(* IEC 61131-3 sources: smart-home/SmartHome/plc (part 2) *)

(* ---- Resource1.gvl ---- *)
(****************************************************************************
**
** Copyright (C) 2021 Francesco Mandracci
** Contact: https://github.com/fmandracci/smart-home
**
** This file is part of the Smart Home Framework.
**
** Commercial License Usage
** Licensees holding valid commercial licenses may use this file in
** accordance with the terms contained in a written agreement
** between you and the copyright owner.
**
** GNU Lesser General Public License Usage
** Alternatively, this file may be used under the terms of the GNU Lesser
** General Public License version 3 as published by the Free Software
** Foundation and appearing in the file LICENSE included in the
** packaging of this file. Please review the following information to
** ensure the GNU Lesser General Public License version 3 requirements
** will be met: https://www.gnu.org/licenses/lgpl-3.0.html.
**
****************************************************************************)

VAR_GLOBAL
    BA_values: ARRAY [1..32] of BOOL;
    BA_masks: ARRAY [1..32] of DWORD := [
        16#00000001,  16#00000002,  16#00000004,  16#00000008,  16#00000010,  16#00000020,  16#00000040,  16#00000080,
        16#00000100,  16#00000200,  16#00000400,  16#00000800,  16#00001000,  16#00002000,  16#00004000,  16#00008000,
        16#00010000,  16#00020000,  16#00040000,  16#00080000,  16#00100000,  16#00200000,  16#00400000,  16#00800000,
        16#01000000,  16#02000000,  16#04000000,  16#08000000,  16#10000000,  16#20000000,  16#40000000,  16#80000000];

END_VAR

(* ---- BA_CheckSensor.st ---- *)
(****************************************************************************
**
** Copyright (C) 2021 Francesco Mandracci
** Contact: https://github.com/fmandracci/smart-home
**
** This file is part of the Smart Home Framework.
**
** Commercial License Usage
** Licensees holding valid commercial licenses may use this file in
** accordance with the terms contained in a written agreement
** between you and the copyright owner.
**
** GNU Lesser General Public License Usage
** Alternatively, this file may be used under the terms of the GNU Lesser
** General Public License version 3 as published by the Free Software
** Foundation and appearing in the file LICENSE included in the
** packaging of this file. Please review the following information to
** ensure the GNU Lesser General Public License version 3 requirements
** will be met: https://www.gnu.org/licenses/lgpl-3.0.html.
**
****************************************************************************)

FUNCTION BA_CheckSensor
#import "Crosstable.gvl"
#import "Resource1.gvl"
VAR_INPUT
	n : UINT;
    konfig : DWORD;
    mask : DWORD;
    PLC_DigIn : BOOL;
END_VAR
VAR_IN_OUT
	ba_ok : UINT;
    all_ok : BOOL;
END_VAR
VAR
	status : UINT;
END_VAR;

	status := ba_ok;

	if PLC_BA_status = ALARM_STATUS_ARMED or PLC_BA_status = ALARM_STATUS_ENABLED
	   or PLC_BA_status = ALARM_STATUS_RINGING or PLC_BA_status = ALARM_STATUS_MUTED then

		(* NB: this function is called only in (ARMED, ENABLED, RINGING, MUTED *)
		if PLC_BA_enabled_sensors >= n then
			if (konfig and mask) <> 0 then
				(* sensor is configured for checking *)

				if PLC_DigIn then
					(* sensor GOOD *)
					if PLC_BA_status = ALARM_STATUS_ARMED then
						status := ALARM_SENSOR_GOOD;
					elsif PLC_BA_status = ALARM_STATUS_ENABLED then
						status := ALARM_SENSOR_GOOD;
					else (* ALARM_STATUS_RINGING or ALARM_STATUS_MUTED *)
						if ba_ok = ALARM_SENSOR_GOOD then
							status := ALARM_SENSOR_GOOD;
						elsif ba_ok = ALARM_SENSOR_NOT_GOOD then
							status := ALARM_SENSOR_WAS_NG;
						else (* ALARM_SENSOR_WAS_NG *)
							status := ALARM_SENSOR_WAS_NG;
						end_if;
					end_if;

				else
					(* sensor NOT GOOD *)
					all_ok := false; (* <--------------------------= *)
					if PLC_BA_status = ALARM_STATUS_ARMED then
						status := ALARM_SENSOR_STILL_NG;
					elsif PLC_BA_status = ALARM_STATUS_ENABLED then
						status := ALARM_SENSOR_NOT_GOOD;
					else (* ALARM_STATUS_RINGING or ALARM_STATUS_MUTED *)
						status := ALARM_SENSOR_NOT_GOOD;
					end_if;
				end_if;
			else
				(* dark grey: sensor is ignored in this bitmask *)
				status := ALARM_SENSOR_IGNORED;
			end_if;
		else
			(* not visible: sensor is not present *)
			status := ALARM_SENSOR_DISABLED;
		end_if;

	end_if;

	if ba_ok <> status then
		ba_ok := status;
	end_if;

END_FUNCTION

(* ---- BA_CheckSensors.st ---- *)
(****************************************************************************
**
** Copyright (C) 2021 Francesco Mandracci
** Contact: https://github.com/fmandracci/smart-home
**
** This file is part of the Smart Home Framework.
**
** Commercial License Usage
** Licensees holding valid commercial licenses may use this file in
** accordance with the terms contained in a written agreement
** between you and the copyright owner.
**
** GNU Lesser General Public License Usage
** Alternatively, this file may be used under the terms of the GNU Lesser
** General Public License version 3 as published by the Free Software
** Foundation and appearing in the file LICENSE included in the
** packaging of this file. Please review the following information to
** ensure the GNU Lesser General Public License version 3 requirements
** will be met: https://www.gnu.org/licenses/lgpl-3.0.html.
**
****************************************************************************)

FUNCTION BA_CheckSensors : BOOL
#import "Crosstable.gvl"
#import "Resource1.gvl"
VAR_INPUT
    index : UINT;
END_VAR
VAR
	mask : UDINT;
	konfig: DWORD;
	all_ok : BOOL;
END_VAR;

	case index of
	ALARM_INDEX_NOTHING: mask := ALARM_MASK_NOTHING;
	ALARM_INDEX_DAYTIME: mask := PLC_BA_daytime_bitmask;
	ALARM_INDEX_NIGHTTIME: mask := PLC_BA_nighttime_bitmask;
	ALARM_INDEX_EVERYTHING: mask := PLC_BA_everything_bitmask;
	else mask := ALARM_MASK_NOTHING;
	end_case;

	konfig := UDINT_TO_DWORD(mask);
	all_ok := true;

    BA_CheckSensor(1 , konfig, 16#00000001, PLC_BA_DigIn_1 , PLC_BA_OK_1 , all_ok);
    BA_CheckSensor(2 , konfig, 16#00000002, PLC_BA_DigIn_2 , PLC_BA_OK_2 , all_ok);
    BA_CheckSensor(3 , konfig, 16#00000004, PLC_BA_DigIn_3 , PLC_BA_OK_3 , all_ok);
    BA_CheckSensor(4 , konfig, 16#00000008, PLC_BA_DigIn_4 , PLC_BA_OK_4 , all_ok);
    BA_CheckSensor(5 , konfig, 16#00000010, PLC_BA_DigIn_5 , PLC_BA_OK_5 , all_ok);
    BA_CheckSensor(6 , konfig, 16#00000020, PLC_BA_DigIn_6 , PLC_BA_OK_6 , all_ok);
    BA_CheckSensor(7 , konfig, 16#00000040, PLC_BA_DigIn_7 , PLC_BA_OK_7 , all_ok);
    BA_CheckSensor(8 , konfig, 16#00000080, PLC_BA_DigIn_8 , PLC_BA_OK_8 , all_ok);
    BA_CheckSensor(9 , konfig, 16#00000100, PLC_BA_DigIn_9 , PLC_BA_OK_9 , all_ok);
    BA_CheckSensor(10, konfig, 16#00000200, PLC_BA_DigIn_10, PLC_BA_OK_10, all_ok);
    BA_CheckSensor(11, konfig, 16#00000400, PLC_BA_DigIn_11, PLC_BA_OK_11, all_ok);
    BA_CheckSensor(12, konfig, 16#00000800, PLC_BA_DigIn_12, PLC_BA_OK_12, all_ok);
    BA_CheckSensor(13, konfig, 16#00001000, PLC_BA_DigIn_13, PLC_BA_OK_13, all_ok);
    BA_CheckSensor(14, konfig, 16#00002000, PLC_BA_DigIn_14, PLC_BA_OK_14, all_ok);
    BA_CheckSensor(15, konfig, 16#00004000, PLC_BA_DigIn_15, PLC_BA_OK_15, all_ok);
    BA_CheckSensor(16, konfig, 16#00008000, PLC_BA_DigIn_16, PLC_BA_OK_16, all_ok);

    BA_CheckSensor(17, konfig, 16#00010000, PLC_BA_DigIn_17, PLC_BA_OK_17, all_ok);
    BA_CheckSensor(18, konfig, 16#00020000, PLC_BA_DigIn_18, PLC_BA_OK_18, all_ok);
    BA_CheckSensor(19, konfig, 16#00040000, PLC_BA_DigIn_19, PLC_BA_OK_19, all_ok);
    BA_CheckSensor(20, konfig, 16#00080000, PLC_BA_DigIn_20, PLC_BA_OK_20, all_ok);
    BA_CheckSensor(21, konfig, 16#00100000, PLC_BA_DigIn_21, PLC_BA_OK_21, all_ok);
    BA_CheckSensor(22, konfig, 16#00200000, PLC_BA_DigIn_22, PLC_BA_OK_22, all_ok);
    BA_CheckSensor(23, konfig, 16#00400000, PLC_BA_DigIn_23, PLC_BA_OK_23, all_ok);
    BA_CheckSensor(24, konfig, 16#00800000, PLC_BA_DigIn_24, PLC_BA_OK_24, all_ok);
    BA_CheckSensor(25, konfig, 16#01000000, PLC_BA_DigIn_25, PLC_BA_OK_25, all_ok);
    BA_CheckSensor(26, konfig, 16#02000000, PLC_BA_DigIn_26, PLC_BA_OK_26, all_ok);
    BA_CheckSensor(27, konfig, 16#04000000, PLC_BA_DigIn_27, PLC_BA_OK_27, all_ok);
    BA_CheckSensor(28, konfig, 16#08000000, PLC_BA_DigIn_28, PLC_BA_OK_28, all_ok);
    BA_CheckSensor(29, konfig, 16#10000000, PLC_BA_DigIn_29, PLC_BA_OK_29, all_ok);
    BA_CheckSensor(30, konfig, 16#20000000, PLC_BA_DigIn_30, PLC_BA_OK_30, all_ok);
    BA_CheckSensor(31, konfig, 16#40000000, PLC_BA_DigIn_31, PLC_BA_OK_31, all_ok);
    BA_CheckSensor(32, konfig, 16#80000000, PLC_BA_DigIn_32, PLC_BA_OK_32, all_ok);

	BA_CheckSensors := all_ok;

END_FUNCTION

(* ---- BA_ClearOK.st ---- *)
(****************************************************************************
**
** Copyright (C) 2021 Francesco Mandracci
** Contact: https://github.com/fmandracci/smart-home
**
** This file is part of the Smart Home Framework.
**
** Commercial License Usage
** Licensees holding valid commercial licenses may use this file in
** accordance with the terms contained in a written agreement
** between you and the copyright owner.
**
** GNU Lesser General Public License Usage
** Alternatively, this file may be used under the terms of the GNU Lesser
** General Public License version 3 as published by the Free Software
** Foundation and appearing in the file LICENSE included in the
** packaging of this file. Please review the following information to
** ensure the GNU Lesser General Public License version 3 requirements
** will be met: https://www.gnu.org/licenses/lgpl-3.0.html.
**
****************************************************************************)

FUNCTION BA_ClearOK : UINT
#import "Crosstable.gvl"
#import "Resource1.gvl"
VAR_INPUT
    n : UINT;
END_VAR

	if PLC_BA_enabled_sensors >= n then
		BA_ClearOK := ALARM_SENSOR_IGNORED;
	else
		BA_ClearOK := ALARM_SENSOR_DISABLED;
	end_if;

END_FUNCTION

(* ---- BA_ClearOKs.st ---- *)
(****************************************************************************
**
** Copyright (C) 2021 Francesco Mandracci
** Contact: https://github.com/fmandracci/smart-home
**
** This file is part of the Smart Home Framework.
**
** Commercial License Usage
** Licensees holding valid commercial licenses may use this file in
** accordance with the terms contained in a written agreement
** between you and the copyright owner.
**
** GNU Lesser General Public License Usage
** Alternatively, this file may be used under the terms of the GNU Lesser
** General Public License version 3 as published by the Free Software
** Foundation and appearing in the file LICENSE included in the
** packaging of this file. Please review the following information to
** ensure the GNU Lesser General Public License version 3 requirements
** will be met: https://www.gnu.org/licenses/lgpl-3.0.html.
**
****************************************************************************)

FUNCTION BA_ClearOKs
#import "Crosstable.gvl"
#import "Resource1.gvl"

    PLC_BA_OK_1  := BA_ClearOK(1 );
    PLC_BA_OK_2  := BA_ClearOK(2 );
    PLC_BA_OK_3  := BA_ClearOK(3 );
    PLC_BA_OK_4  := BA_ClearOK(4 );
    PLC_BA_OK_5  := BA_ClearOK(5 );
    PLC_BA_OK_6  := BA_ClearOK(6 );
    PLC_BA_OK_7  := BA_ClearOK(7 );
    PLC_BA_OK_8  := BA_ClearOK(8 );
    PLC_BA_OK_9  := BA_ClearOK(9 );
    PLC_BA_OK_10 := BA_ClearOK(10);
    PLC_BA_OK_11 := BA_ClearOK(11);
    PLC_BA_OK_12 := BA_ClearOK(12);
    PLC_BA_OK_13 := BA_ClearOK(13);
    PLC_BA_OK_14 := BA_ClearOK(14);
    PLC_BA_OK_15 := BA_ClearOK(15);
    PLC_BA_OK_16 := BA_ClearOK(16);

    PLC_BA_OK_17 := BA_ClearOK(17);
    PLC_BA_OK_18 := BA_ClearOK(18);
    PLC_BA_OK_19 := BA_ClearOK(19);
    PLC_BA_OK_20 := BA_ClearOK(20);
    PLC_BA_OK_21 := BA_ClearOK(21);
    PLC_BA_OK_22 := BA_ClearOK(22);
    PLC_BA_OK_23 := BA_ClearOK(23);
    PLC_BA_OK_24 := BA_ClearOK(24);
    PLC_BA_OK_25 := BA_ClearOK(25);
    PLC_BA_OK_26 := BA_ClearOK(26);
    PLC_BA_OK_27 := BA_ClearOK(27);
    PLC_BA_OK_28 := BA_ClearOK(28);
    PLC_BA_OK_29 := BA_ClearOK(29);
    PLC_BA_OK_30 := BA_ClearOK(30);
    PLC_BA_OK_31 := BA_ClearOK(31);
    PLC_BA_OK_32 := BA_ClearOK(32);

END_FUNCTION

(* ---- BA_ReadSensor.st ---- *)
(****************************************************************************
**
** Copyright (C) 2021 Francesco Mandracci
** Contact: https://github.com/fmandracci/smart-home
**
** This file is part of the Smart Home Framework.
**
** Commercial License Usage
** Licensees holding valid commercial licenses may use this file in
** accordance with the terms contained in a written agreement
** between you and the copyright owner.
**
** GNU Lesser General Public License Usage
** Alternatively, this file may be used under the terms of the GNU Lesser
** General Public License version 3 as published by the Free Software
** Foundation and appearing in the file LICENSE included in the
** packaging of this file. Please review the following information to
** ensure the GNU Lesser General Public License version 3 requirements
** will be met: https://www.gnu.org/licenses/lgpl-3.0.html.
**
****************************************************************************)

FUNCTION BA_ReadSensor : BOOL
#import "Crosstable.gvl"
#import "Resource1.gvl"
VAR_INPUT
    n : UINT;
END_VAR

	if PLC_BA_enabled_sensors >= n then

		if PLC_control_type = ControlType_2 then
			(* MPNE_A, MPNE_B on RTU0 *)
			if n <= 16 then
				if NODE_11_STATUS = NODE_NODE_OK then
					case n of
		             1: SetMpneDigDir_IN(MPNE_A_DigDir_1); BA_ReadSensor := MPNE_A_DigIn_1 ;
		             2: SetMpneDigDir_IN(MPNE_A_DigDir_2); BA_ReadSensor := MPNE_A_DigIn_2 ;
		             3: SetMpneDigDir_IN(MPNE_A_DigDir_3); BA_ReadSensor := MPNE_A_DigIn_3 ;
		             4: SetMpneDigDir_IN(MPNE_A_DigDir_4); BA_ReadSensor := MPNE_A_DigIn_4 ;
		             5: SetMpneDigDir_IN(MPNE_A_DigDir_5); BA_ReadSensor := MPNE_A_DigIn_5 ;
		             6: SetMpneDigDir_IN(MPNE_A_DigDir_6); BA_ReadSensor := MPNE_A_DigIn_6 ;
		             7: SetMpneDigDir_IN(MPNE_A_DigDir_7); BA_ReadSensor := MPNE_A_DigIn_7 ;
		             8: SetMpneDigDir_IN(MPNE_A_DigDir_8); BA_ReadSensor := MPNE_A_DigIn_8 ;
		             9:                                    BA_ReadSensor := MPNE_A_DigIn_9 ;
		            10:                                    BA_ReadSensor := MPNE_A_DigIn_10;
		            11:                                    BA_ReadSensor := MPNE_A_DigIn_11;
		            12:                                    BA_ReadSensor := MPNE_A_DigIn_12;
		            13:                                    BA_ReadSensor := MPNE_A_DigIn_13;
		            14:                                    BA_ReadSensor := MPNE_A_DigIn_14;
		            15:                                    BA_ReadSensor := MPNE_A_DigIn_15;
		            16:                                    BA_ReadSensor := MPNE_A_DigIn_16;
					else
						BA_ReadSensor := false;
					end_case;
				else
					BA_ReadSensor := false;
				end_if;
			else
				if NODE_12_STATUS = NODE_NODE_OK then
					case n of
		            17: SetMpneDigDir_IN(MPNE_B_DigDir_1); BA_ReadSensor := MPNE_B_DigIn_1 ;
		            18: SetMpneDigDir_IN(MPNE_B_DigDir_2); BA_ReadSensor := MPNE_B_DigIn_2 ;
		            19: SetMpneDigDir_IN(MPNE_B_DigDir_3); BA_ReadSensor := MPNE_B_DigIn_3 ;
		            20: SetMpneDigDir_IN(MPNE_B_DigDir_4); BA_ReadSensor := MPNE_B_DigIn_4 ;
		            21: SetMpneDigDir_IN(MPNE_B_DigDir_5); BA_ReadSensor := MPNE_B_DigIn_5 ;
		            22: SetMpneDigDir_IN(MPNE_B_DigDir_6); BA_ReadSensor := MPNE_B_DigIn_6 ;
		            23: SetMpneDigDir_IN(MPNE_B_DigDir_7); BA_ReadSensor := MPNE_B_DigIn_7 ;
		            24: SetMpneDigDir_IN(MPNE_B_DigDir_8); BA_ReadSensor := MPNE_B_DigIn_8 ;

		            25:                                    BA_ReadSensor := MPNE_B_DigIn_9 ;
		            26:                                    BA_ReadSensor := MPNE_B_DigIn_10;
		            27:                                    BA_ReadSensor := MPNE_B_DigIn_11;
		            28:                                    BA_ReadSensor := MPNE_B_DigIn_12;
		            29:                                    BA_ReadSensor := MPNE_B_DigIn_13;
		            30:                                    BA_ReadSensor := MPNE_B_DigIn_14;
		            31:                                    BA_ReadSensor := MPNE_B_DigIn_15;
		            32:                                    BA_ReadSensor := MPNE_B_DigIn_16;
					else BA_ReadSensor := false;
					end_case;
				else
					BA_ReadSensor := false;
				end_if;
			end_if;

		elsif PLC_control_type = ControlType_7 then
			(* Fast I/O on GPIO *)
			case n of
             1: BA_ReadSensor := PLC_FastIO_1 ;
             2: BA_ReadSensor := PLC_FastIO_2 ;
             3: BA_ReadSensor := PLC_FastIO_3 ;
			else BA_ReadSensor := false;
			end_case;

		elsif PLC_control_type = ControlType_12 then
			(* Fast I/O on GPIO *)
			case n of
             1: BA_ReadSensor := PLC_FastIO_1 ;
             2: BA_ReadSensor := PLC_FastIO_2 ;
             3: BA_ReadSensor := PLC_FastIO_3 ;
			else BA_ReadSensor := false;
			end_case;

		elsif PLC_control_type = ControlType_13 then
			(* TPAC1007_04_AD Local I/O on RTU3 *)
			if NODE_31_STATUS = NODE_NODE_OK then
				case n of
	             1: BA_ReadSensor := PLC_DigIn_9 ;
	             2: BA_ReadSensor := PLC_DigIn_10;
	             3: BA_ReadSensor := PLC_DigIn_11;
				else BA_ReadSensor := false;
				end_case;
			else BA_ReadSensor := false;
			end_if;

		elsif PLC_control_type = ControlType_14 or PLC_control_type = ControlType_6 then
			(* MPNC DI16 "A,B" + DO16 "A,B" on RTU0 *)
			if NODE_27_STATUS = NODE_NODE_OK then
				case n of
	             1: BA_ReadSensor := MPNC_DigIn_A_1 ;
	             2: BA_ReadSensor := MPNC_DigIn_A_2 ;
	             3: BA_ReadSensor := MPNC_DigIn_A_3 ;
	             4: BA_ReadSensor := MPNC_DigIn_A_4 ;
	             5: BA_ReadSensor := MPNC_DigIn_A_5 ;
	             6: BA_ReadSensor := MPNC_DigIn_A_6 ;
	             7: BA_ReadSensor := MPNC_DigIn_A_7 ;
	             8: BA_ReadSensor := MPNC_DigIn_A_8 ;
	             9: BA_ReadSensor := MPNC_DigIn_A_9 ;
	            10: BA_ReadSensor := MPNC_DigIn_A_10;
	            11: BA_ReadSensor := MPNC_DigIn_A_11;
	            12: BA_ReadSensor := MPNC_DigIn_A_12;
	            13: BA_ReadSensor := MPNC_DigIn_A_13;
	            14: BA_ReadSensor := MPNC_DigIn_A_14;
	            15: BA_ReadSensor := MPNC_DigIn_A_15;
	            16: BA_ReadSensor := MPNC_DigIn_A_16;

	            17: BA_ReadSensor := MPNC_DigIn_B_1 ;
	            18: BA_ReadSensor := MPNC_DigIn_B_2 ;
	            19: BA_ReadSensor := MPNC_DigIn_B_3 ;
	            20: BA_ReadSensor := MPNC_DigIn_B_4 ;
	            21: BA_ReadSensor := MPNC_DigIn_B_5 ;
	            22: BA_ReadSensor := MPNC_DigIn_B_6 ;
	            23: BA_ReadSensor := MPNC_DigIn_B_7 ;
	            24: BA_ReadSensor := MPNC_DigIn_B_8 ;
	            25: BA_ReadSensor := MPNC_DigIn_B_9 ;
	            26: BA_ReadSensor := MPNC_DigIn_B_10;
	            27: BA_ReadSensor := MPNC_DigIn_B_11;
	            28: BA_ReadSensor := MPNC_DigIn_B_12;
	            29: BA_ReadSensor := MPNC_DigIn_B_13;
	            30: BA_ReadSensor := MPNC_DigIn_B_14;
	            31: BA_ReadSensor := MPNC_DigIn_B_15;
	            32: BA_ReadSensor := MPNC_DigIn_B_16;
	            else BA_ReadSensor := false;
				end_case;
			else BA_ReadSensor := false;
			end_if;

		end_if;

	else
		BA_ReadSensor := false;

	end_if;

END_FUNCTION

(* ---- BA_ReadSensors.st ---- *)
(****************************************************************************
**
** Copyright (C) 2021 Francesco Mandracci
** Contact: https://github.com/fmandracci/smart-home
**
** This file is part of the Smart Home Framework.
**
** Commercial License Usage
** Licensees holding valid commercial licenses may use this file in
** accordance with the terms contained in a written agreement
** between you and the copyright owner.
**
** GNU Lesser General Public License Usage
** Alternatively, this file may be used under the terms of the GNU Lesser
** General Public License version 3 as published by the Free Software
** Foundation and appearing in the file LICENSE included in the
** packaging of this file. Please review the following information to
** ensure the GNU Lesser General Public License version 3 requirements
** will be met: https://www.gnu.org/licenses/lgpl-3.0.html.
**
****************************************************************************)

FUNCTION BA_ReadSensors
#import "Crosstable.gvl"
#import "Resource1.gvl"

		(* 1/2 alarm sensors *)

        PLC_BA_DigIn_1 := BA_ReadSensor(1 );
        PLC_BA_DigIn_2 := BA_ReadSensor(2 );
        PLC_BA_DigIn_3 := BA_ReadSensor(3 );
        PLC_BA_DigIn_4 := BA_ReadSensor(4 );
        PLC_BA_DigIn_5 := BA_ReadSensor(5 );
        PLC_BA_DigIn_6 := BA_ReadSensor(6 );
        PLC_BA_DigIn_7 := BA_ReadSensor(7 );
        PLC_BA_DigIn_8 := BA_ReadSensor(8 );

        PLC_BA_DigIn_9 := BA_ReadSensor(9 );
        PLC_BA_DigIn_10:= BA_ReadSensor(10);
        PLC_BA_DigIn_11:= BA_ReadSensor(11);
        PLC_BA_DigIn_12:= BA_ReadSensor(12);
        PLC_BA_DigIn_13:= BA_ReadSensor(13);
        PLC_BA_DigIn_14:= BA_ReadSensor(14);
        PLC_BA_DigIn_15:= BA_ReadSensor(15);
        PLC_BA_DigIn_16:= BA_ReadSensor(16);

        PLC_BA_DigIn_17:= BA_ReadSensor(17);
        PLC_BA_DigIn_18:= BA_ReadSensor(18);
        PLC_BA_DigIn_19:= BA_ReadSensor(19);
        PLC_BA_DigIn_20:= BA_ReadSensor(20);
        PLC_BA_DigIn_21:= BA_ReadSensor(21);
        PLC_BA_DigIn_22:= BA_ReadSensor(22);
        PLC_BA_DigIn_23:= BA_ReadSensor(23);
        PLC_BA_DigIn_24:= BA_ReadSensor(24);

        PLC_BA_DigIn_25:= BA_ReadSensor(25);
        PLC_BA_DigIn_26:= BA_ReadSensor(26);
        PLC_BA_DigIn_27:= BA_ReadSensor(27);
        PLC_BA_DigIn_28:= BA_ReadSensor(28);
        PLC_BA_DigIn_29:= BA_ReadSensor(29);
        PLC_BA_DigIn_30:= BA_ReadSensor(30);
        PLC_BA_DigIn_31:= BA_ReadSensor(31);
        PLC_BA_DigIn_32:= BA_ReadSensor(32);

		(* 2/2 other sensors (blackout detection, ...) *)

		if PLC_control_type = ControlType_2 then
			(* MPNE_A, MPNE_B on RTU0 *)
			if PLC_PRODUCT_ID = 16#100704AD or PLC_PRODUCT_ID = 16#100704AA or PLC_PRODUCT_ID = 16#100704AC then
				PLC_BA_input_9  := PLC_DigIn_9 ;
			    PLC_BA_input_10 := PLC_DigIn_10;
			    PLC_BA_input_11 := PLC_DigIn_11;
				PLC_BA_input_12 := PLC_DigIn_12;
				PLC_BA_blackout_digin := PLC_DigIn_12; (* --> PLC_BA_BlackoutDetected Alarm *)
			elsif  PLC_PRODUCT_ID = 16#1043030C then
				PLC_BA_input_9  := PLC_FastIO_1 ;
			    PLC_BA_input_10 := PLC_FastIO_2;
			    PLC_BA_input_11 := PLC_FastIO_3;
				PLC_BA_input_12 := PLC_FastIO_4;
				PLC_BA_blackout_digin := PLC_FastIO_4; (* --> PLC_BA_BlackoutDetected Alarm *)
			else (* 16#100704AE *)
				PLC_BA_input_9  := false;
			    PLC_BA_input_10 := false;
			    PLC_BA_input_11 := false;
				PLC_BA_input_12 := false;
				PLC_BA_blackout_digin := false; (* --> PLC_BA_BlackoutDetected Alarm *)
			end_if;

		elsif PLC_control_type = ControlType_7 then
			(* Fast I/O on GPIO *)
			PLC_BA_input_9  := false;
		    PLC_BA_input_10 := false;
		    PLC_BA_input_11 := false;
			PLC_BA_input_12 := PLC_FastIO_4;
			PLC_BA_blackout_digin := PLC_FastIO_4; (* --> PLC_BA_BlackoutDetected Alarm *)

		elsif PLC_control_type = ControlType_12 then
			(* Fast I/O on GPIO *)
			PLC_BA_input_9  := false;
		    PLC_BA_input_10 := false;
		    PLC_BA_input_11 := false;
			PLC_BA_input_12 := PLC_FastIO_4;
			PLC_BA_blackout_digin := PLC_FastIO_4; (* --> PLC_BA_BlackoutDetected Alarm *)

		elsif PLC_control_type = ControlType_13 then
			(* TPAC1007_04_AD Local I/O on RTU3 *)
			PLC_BA_input_9  := PLC_DigIn_9 ;
		    PLC_BA_input_10 := PLC_DigIn_10;
		    PLC_BA_input_11 := PLC_DigIn_11;
			PLC_BA_input_12 := PLC_DigIn_12;
			PLC_BA_blackout_digin := PLC_DigIn_12; (* --> PLC_BA_BlackoutDetected Alarm *)

		elsif PLC_control_type = ControlType_14 or PLC_control_type = ControlType_6 then
			(* MPNC DI16 "A,B" + DO16 "A,B" on RTU0 *)
			PLC_BA_input_9  := false ;
		    PLC_BA_input_10 := false;
		    PLC_BA_input_11 := false;
			PLC_BA_input_12 := false;
			PLC_BA_blackout_digin := false; (* --> PLC_BA_BlackoutDetected Alarm *)

		end_if;

END_FUNCTION

(* ---- BA_ReadSensorsReady.st ---- *)
(****************************************************************************
**
** Copyright (C) 2021 Francesco Mandracci
** Contact: https://github.com/fmandracci/smart-home
**
** This file is part of the Smart Home Framework.
**
** Commercial License Usage
** Licensees holding valid commercial licenses may use this file in
** accordance with the terms contained in a written agreement
** between you and the copyright owner.
**
** GNU Lesser General Public License Usage
** Alternatively, this file may be used under the terms of the GNU Lesser
** General Public License version 3 as published by the Free Software
** Foundation and appearing in the file LICENSE included in the
** packaging of this file. Please review the following information to
** ensure the GNU Lesser General Public License version 3 requirements
** will be met: https://www.gnu.org/licenses/lgpl-3.0.html.
**
****************************************************************************)

FUNCTION BA_ReadSensorsReady : BOOL
#import "Crosstable.gvl"
#import "Resource1.gvl"

	if PLC_control_type = ControlType_2 then
		(* MPNE_A, MPNE_B on RTU0 *)

		if PLC_BA_enabled_sensors <= 16 then
			BA_ReadSensorsReady := (NODE_11_STATUS = NODE_NODE_OK);
		else
			BA_ReadSensorsReady := (NODE_11_STATUS = NODE_NODE_OK) and (NODE_12_STATUS = NODE_NODE_OK);
		end_if;

	elsif PLC_control_type = ControlType_7 then
		(* Fast I/O on GPIO *)
		BA_ReadSensorsReady := true;

	elsif PLC_control_type = ControlType_9 then
		(* MPNE_E on RTU3 *)
		BA_ReadSensorsReady :=  (NODE_45_STATUS = NODE_NODE_OK);

	elsif PLC_control_type = ControlType_99 then
		(* MPNE_A on RTU0 *)
		BA_ReadSensorsReady :=  (NODE_11_STATUS = NODE_NODE_OK);

	elsif PLC_control_type = ControlType_12 then
		(* Fast I/O on GPIO *)
		BA_ReadSensorsReady := true;

	elsif PLC_control_type = ControlType_13 then
		(* TPAC1007_04_AD Local I/O on RTU3 *)
		BA_ReadSensorsReady := (NODE_31_STATUS = NODE_NODE_OK);

	elsif PLC_control_type = ControlType_16 then
		(* TPAC1007_04_AD Local I/O on RTU3 *)
		BA_ReadSensorsReady := (NODE_31_STATUS = NODE_NODE_OK);

	elsif PLC_control_type = ControlType_14 or PLC_control_type = ControlType_6 then
		(* MPNC DI16 "A,B" + DO16 "A,B" on RTU0 *)
		BA_ReadSensorsReady := (NODE_27_STATUS = NODE_NODE_OK);

	else
		BA_ReadSensorsReady := false;

	end_if;

END_FUNCTION

(* ---- BA_SetDigOuts.st ---- *)
(****************************************************************************
**
** Copyright (C) 2021 Francesco Mandracci
** Contact: https://github.com/fmandracci/smart-home
**
** This file is part of the Smart Home Framework.
**
** Commercial License Usage
** Licensees holding valid commercial licenses may use this file in
** accordance with the terms contained in a written agreement
** between you and the copyright owner.
**
** GNU Lesser General Public License Usage
** Alternatively, this file may be used under the terms of the GNU Lesser
** General Public License version 3 as published by the Free Software
** Foundation and appearing in the file LICENSE included in the
** packaging of this file. Please review the following information to
** ensure the GNU Lesser General Public License version 3 requirements
** will be met: https://www.gnu.org/licenses/lgpl-3.0.html.
**
****************************************************************************)

FUNCTION BA_SetDigOuts
#import "Crosstable.gvl"
#import "Resource1.gvl"
VAR_INPUT
	green    : BOOL;
	red      : BOOL;
	yellow1  : BOOL;
	yellow2  : BOOL;

	siren    : BOOL;
	enable_A : BOOL;
	enable_B : BOOL;
	enable_C : BOOL;
END_VAR

	if PLC_control_type = ControlType_2 then
		if PLC_PRODUCT_ID = 16#100704AD or PLC_PRODUCT_ID = 16#100704AA or PLC_PRODUCT_ID = 16#100704AC then
			(* sensors: MPNE_A, MPNE_B on RTU0; leds: TPAC1007_04_AD/AA/AC Local I/O on RTU3 *)

        	if PLC_DigDir_1 <> DigDir_OUT then PLC_DigDir_1 := DigDir_OUT; end_if;
        	if PLC_DigDir_2 <> DigDir_OUT then PLC_DigDir_2 := DigDir_OUT; end_if;
        	if PLC_DigDir_3 <> DigDir_OUT then PLC_DigDir_3 := DigDir_OUT; end_if;
        	if PLC_DigDir_4 <> DigDir_OUT then PLC_DigDir_4 := DigDir_OUT; end_if;

        	if PLC_DigDir_5 <> DigDir_OUT then PLC_DigDir_5 := DigDir_OUT; end_if;
        	if PLC_DigDir_6 <> DigDir_OUT then PLC_DigDir_6 := DigDir_OUT; end_if;
        	if PLC_DigDir_7 <> DigDir_OUT then PLC_DigDir_7 := DigDir_OUT; end_if;
        	if PLC_DigDir_8 <> DigDir_OUT then PLC_DigDir_8 := DigDir_OUT; end_if;

	        if PLC_DigOut_1 <> green    then PLC_DigOut_1 := green   ; end_if;
	        if PLC_DigOut_2 <> red      then PLC_DigOut_2 := red     ; end_if;
	        if PLC_DigOut_3 <> yellow1  then PLC_DigOut_3 := yellow1 ; end_if;
	        if PLC_DigOut_4 <> yellow2  then PLC_DigOut_4 := yellow2 ; end_if;

	        if PLC_DigOut_5 <> siren    then PLC_DigOut_5 := siren   ; end_if;
	        if PLC_DigOut_6 <> enable_A then PLC_DigOut_6 := enable_A; end_if;
	        if PLC_DigOut_7 <> enable_B then PLC_DigOut_7 := enable_B; end_if;
	        if PLC_DigOut_8 <> enable_C then PLC_DigOut_8 := enable_C; end_if;

		elsif PLC_PRODUCT_ID = 16#100704AE then
			(* sensors: MPNE_A, MPNE_B on RTU0; leds: TPAC1007_04_AE Local I/O on RTU3 *)
        	if PLC_DigDir_1 <> DigDir_OUT then PLC_DigDir_1 := DigDir_OUT; end_if;
        	if PLC_DigDir_2 <> DigDir_OUT then PLC_DigDir_2 := DigDir_OUT; end_if;
        	if PLC_DigDir_3 <> DigDir_OUT then PLC_DigDir_3 := DigDir_OUT; end_if;
        	if PLC_DigDir_4 <> DigDir_OUT then PLC_DigDir_4 := DigDir_OUT; end_if;

        	if PLC_DigDir_5 <> DigDir_OUT then PLC_DigDir_5 := DigDir_OUT; end_if;
        	if PLC_DigDir_6 <> DigDir_OUT then PLC_DigDir_6 := DigDir_OUT; end_if;
        	if PLC_DigDir_7 <> DigDir_OUT then PLC_DigDir_7 := DigDir_OUT; end_if;
        	if PLC_DigDir_8 <> DigDir_OUT then PLC_DigDir_8 := DigDir_OUT; end_if;

            if getBit(PLC_AnInConf_1, 16#0001) <> green    then setBit(16#0001, green   , PLC_AnInConf_1); end_if;
            if getBit(PLC_AnInConf_1, 16#0002) <> red      then setBit(16#0002, red     , PLC_AnInConf_1); end_if;
            if getBit(PLC_AnInConf_1, 16#0004) <> yellow1  then setBit(16#0004, yellow1 , PLC_AnInConf_1); end_if;
            if getBit(PLC_AnInConf_1, 16#0008) <> yellow2  then setBit(16#0008, yellow2 , PLC_AnInConf_1); end_if;

            if getBit(PLC_AnInConf_1, 16#0010) <> siren    then setBit(16#0010, siren   , PLC_AnInConf_1); end_if;
            if getBit(PLC_AnInConf_1, 16#0020) <> enable_A then setBit(16#0020, enable_A, PLC_AnInConf_1); end_if;
            if getBit(PLC_AnInConf_1, 16#0040) <> enable_B then setBit(16#0040, enable_B, PLC_AnInConf_1); end_if;
            if getBit(PLC_AnInConf_1, 16#0080) <> enable_C then setBit(16#0080, enable_C, PLC_AnInConf_1); end_if;

	    elsif PLC_PRODUCT_ID = 16#1043030C then
			(* sensors: MPNE_A, MPNE_B on RTU0; leds: Fast I/O on GPIO *)
			(* no leds *)
	        if PLC_FastIO_5 <> siren    then PLC_FastIO_5 := siren   ; end_if;
	        if PLC_FastIO_6 <> enable_A then PLC_FastIO_6 := enable_A; end_if;
	        if PLC_FastIO_7 <> enable_B then PLC_FastIO_7 := enable_B; end_if;
	        if PLC_FastIO_8 <> enable_C then PLC_FastIO_8 := enable_C; end_if;

		end_if;

	elsif PLC_control_type = ControlType_7 then
		(* Fast I/O on GPIO *)
		(* no leds, all enabled in one DigOut *)
        if PLC_FastIO_5 <> siren                              then PLC_FastIO_5 := siren                             ; end_if;
        if PLC_FastIO_6 <> (enable_A or enable_B or enable_C) then PLC_FastIO_6 := (enable_A or enable_B or enable_C); end_if;

	elsif PLC_control_type = ControlType_12 then
		(* Fast I/O on GPIO *)
		(* no leds, all enabled in one DigOut *)
        if PLC_FastIO_5 <> siren                              then PLC_FastIO_5 := siren                             ; end_if;
        if PLC_FastIO_6 <> (enable_A or enable_B or enable_C) then PLC_FastIO_6 := (enable_A or enable_B or enable_C); end_if;

	elsif PLC_control_type = ControlType_13 then
		(* TPAC1007_04_AD Local I/O on RTU3 *)
		(* no leds, all enabled in one DigOut *)
    	if PLC_DigDir_5 <> DigDir_OUT then PLC_DigDir_5 := DigDir_OUT; end_if;
    	if PLC_DigDir_6 <> DigDir_OUT then PLC_DigDir_6 := DigDir_OUT; end_if;

        if PLC_DigOut_5 <> siren                              then PLC_DigOut_5 := siren                             ; end_if;
        if PLC_DigOut_6 <> (enable_A or enable_B or enable_C) then PLC_DigOut_6 := (enable_A or enable_B or enable_C); end_if;

	elsif PLC_control_type = ControlType_6 then
		; (* no leds nor digouts *)

	elsif PLC_control_type = ControlType_14 then
		(* MPNC DI16 "A,B" + DO16 "A,B" on RTU0; leds on base DO *)
		(* no leds*)

    	if MPNC_DigDir_5 <> DigDir_OUT then MPNC_DigDir_5 := DigDir_OUT; end_if;
    	if MPNC_DigDir_6 <> DigDir_OUT then MPNC_DigDir_6 := DigDir_OUT; end_if;
    	if MPNC_DigDir_7 <> DigDir_OUT then MPNC_DigDir_7 := DigDir_OUT; end_if;
    	if MPNC_DigDir_8 <> DigDir_OUT then MPNC_DigDir_8 := DigDir_OUT; end_if;

        if MPNC_DigOut_5 <> siren    then MPNC_DigOut_5 := siren   ; end_if;
        if MPNC_DigOut_6 <> enable_A then MPNC_DigOut_6 := enable_A; end_if;
        if MPNC_DigOut_7 <> enable_B then MPNC_DigOut_7 := enable_B; end_if;
        if MPNC_DigOut_8 <> enable_C then MPNC_DigOut_8 := enable_C; end_if;

	end_if;

END_FUNCTION

(* ---- BA_TestConfig.st ---- *)
(****************************************************************************
**
** Copyright (C) 2021 Francesco Mandracci
** Contact: https://github.com/fmandracci/smart-home
**
** This file is part of the Smart Home Framework.
**
** Commercial License Usage
** Licensees holding valid commercial licenses may use this file in
** accordance with the terms contained in a written agreement
** between you and the copyright owner.
**
** GNU Lesser General Public License Usage
** Alternatively, this file may be used under the terms of the GNU Lesser
** General Public License version 3 as published by the Free Software
** Foundation and appearing in the file LICENSE included in the
** packaging of this file. Please review the following information to
** ensure the GNU Lesser General Public License version 3 requirements
** will be met: https://www.gnu.org/licenses/lgpl-3.0.html.
**
****************************************************************************)

FUNCTION BA_TestConfig
#import "Crosstable.gvl"
#import "Resource1.gvl"

    BA_values[ 1] := PLC_BA_DigOut_1 ;
    BA_values[ 2] := PLC_BA_DigOut_2 ;
    BA_values[ 3] := PLC_BA_DigOut_3 ;
    BA_values[ 4] := PLC_BA_DigOut_4 ;
    BA_values[ 5] := PLC_BA_DigOut_5 ;
    BA_values[ 6] := PLC_BA_DigOut_6 ;
    BA_values[ 7] := PLC_BA_DigOut_7 ;
    BA_values[ 8] := PLC_BA_DigOut_8 ;

    BA_values[ 9] := PLC_BA_DigOut_9 ;
    BA_values[10] := PLC_BA_DigOut_10;
    BA_values[11] := PLC_BA_DigOut_11;
    BA_values[12] := PLC_BA_DigOut_12;
    BA_values[13] := PLC_BA_DigOut_13;
    BA_values[14] := PLC_BA_DigOut_14;
    BA_values[15] := PLC_BA_DigOut_15;
    BA_values[16] := PLC_BA_DigOut_16;

    BA_values[17] := PLC_BA_DigOut_17;
    BA_values[18] := PLC_BA_DigOut_18;
    BA_values[19] := PLC_BA_DigOut_19;
    BA_values[20] := PLC_BA_DigOut_20;
    BA_values[21] := PLC_BA_DigOut_21;
    BA_values[22] := PLC_BA_DigOut_22;
    BA_values[23] := PLC_BA_DigOut_23;
    BA_values[24] := PLC_BA_DigOut_24;

    BA_values[25] := PLC_BA_DigOut_25;
    BA_values[26] := PLC_BA_DigOut_26;
    BA_values[27] := PLC_BA_DigOut_27;
    BA_values[28] := PLC_BA_DigOut_28;
    BA_values[29] := PLC_BA_DigOut_29;
    BA_values[30] := PLC_BA_DigOut_30;
    BA_values[31] := PLC_BA_DigOut_31;
    BA_values[32] := PLC_BA_DigOut_32;

    BA_WriteConfigBits(BA_values);

END_FUNCTION

(* ---- BA_Watchdog.st ---- *)
(****************************************************************************
**
** Copyright (C) 2021 Francesco Mandracci
** Contact: https://github.com/fmandracci/smart-home
**
** This file is part of the Smart Home Framework.
**
** Commercial License Usage
** Licensees holding valid commercial licenses may use this file in
** accordance with the terms contained in a written agreement
** between you and the copyright owner.
**
** GNU Lesser General Public License Usage
** Alternatively, this file may be used under the terms of the GNU Lesser
** General Public License version 3 as published by the Free Software
** Foundation and appearing in the file LICENSE included in the
** packaging of this file. Please review the following information to
** ensure the GNU Lesser General Public License version 3 requirements
** will be met: https://www.gnu.org/licenses/lgpl-3.0.html.
**
****************************************************************************)

FUNCTION BA_Watchdog
#import "Crosstable.gvl"
#import "Resource1.gvl"

	if PLC_control_type = ControlType_2 then
		(* MPNE_A, MPNE_B on RTU0 *)
		if (PLC_BA_enabled_sensors >=  1) then
			if MPNE_A_Watchdog <> WatchDogTimeout_s and NODE_11_STATUS = NODE_NODE_OK then
				MPNE_A_Watchdog := WatchDogTimeout_s;
			end_if;
		end_if;
        if (PLC_BA_enabled_sensors >= 17) then
			if MPNE_B_Watchdog <> WatchDogTimeout_s and NODE_12_STATUS = NODE_NODE_OK then
				MPNE_B_Watchdog := WatchDogTimeout_s;
			end_if;
		end_if;

	elsif PLC_control_type = ControlType_7 then
		; (* Fast I/O on GPIO *)

	elsif PLC_control_type = ControlType_12 then
		; (* Fast I/O on GPIO *)

	elsif PLC_control_type = ControlType_13 then
		; (* TPAC1007_04_AD Local I/O on RTU3 *)

	elsif PLC_control_type = ControlType_14 or PLC_control_type = ControlType_6 then
		(* MPNC DI16 "A,B" + DO16 "A,B" on RTU0 *)
		if MPNC_WatchDog <> WatchDogTimeout_s and NODE_27_STATUS = NODE_NODE_OK then
			MPNC_WatchDog := WatchDogTimeout_s;
		end_if;
	end_if;

END_FUNCTION

(* ---- BA_WriteConfig.st ---- *)
(****************************************************************************
**
** Copyright (C) 2021 Francesco Mandracci
** Contact: https://github.com/fmandracci/smart-home
**
** This file is part of the Smart Home Framework.
**
** Commercial License Usage
** Licensees holding valid commercial licenses may use this file in
** accordance with the terms contained in a written agreement
** between you and the copyright owner.
**
** GNU Lesser General Public License Usage
** Alternatively, this file may be used under the terms of the GNU Lesser
** General Public License version 3 as published by the Free Software
** Foundation and appearing in the file LICENSE included in the
** packaging of this file. Please review the following information to
** ensure the GNU Lesser General Public License version 3 requirements
** will be met: https://www.gnu.org/licenses/lgpl-3.0.html.
**
****************************************************************************)

FUNCTION BA_WriteConfig
#import "Crosstable.gvl"
#import "Resource1.gvl"
VAR_INPUT
    index : UINT;
END_VAR
VAR_OUTPUT
    config_index : UINT;
    config_mask : UDINT;
END_VAR
VAR
    n : UINT;
    mask : UDINT;
    konfig: DWORD;
END_VAR

    case index of
    ALARM_INDEX_NOTHING:    mask := ALARM_MASK_NOTHING;
    ALARM_INDEX_DAYTIME:    mask := PLC_BA_daytime_bitmask;
    ALARM_INDEX_NIGHTTIME:  mask := PLC_BA_nighttime_bitmask;
    ALARM_INDEX_EVERYTHING: mask := PLC_BA_everything_bitmask;
    else                    mask := ALARM_MASK_NOTHING;
    end_case;

    config_index := index;
    config_mask := mask;
    konfig := UDINT_TO_DWORD(mask);
    for n := 1 to 32 BY 1 do
        BA_values[n] := (konfig and BA_masks[n]) <> 0;
    end_for;

    BA_WriteConfigBits(BA_values);

    PLC_BA_DigOut_1  := BA_values[ 1];
    PLC_BA_DigOut_2  := BA_values[ 2];
    PLC_BA_DigOut_3  := BA_values[ 3];
    PLC_BA_DigOut_4  := BA_values[ 4];
    PLC_BA_DigOut_5  := BA_values[ 5];
    PLC_BA_DigOut_6  := BA_values[ 6];
    PLC_BA_DigOut_7  := BA_values[ 7];
    PLC_BA_DigOut_8  := BA_values[ 8];

    PLC_BA_DigOut_9  := BA_values[ 9];
    PLC_BA_DigOut_10 := BA_values[10];
    PLC_BA_DigOut_11 := BA_values[11];
    PLC_BA_DigOut_12 := BA_values[12];
    PLC_BA_DigOut_13 := BA_values[13];
    PLC_BA_DigOut_14 := BA_values[14];
    PLC_BA_DigOut_15 := BA_values[15];
    PLC_BA_DigOut_16 := BA_values[16];

    PLC_BA_DigOut_17 := BA_values[17];
    PLC_BA_DigOut_18 := BA_values[18];
    PLC_BA_DigOut_19 := BA_values[19];
    PLC_BA_DigOut_20 := BA_values[20];
    PLC_BA_DigOut_21 := BA_values[21];
    PLC_BA_DigOut_22 := BA_values[22];
    PLC_BA_DigOut_23 := BA_values[23];
    PLC_BA_DigOut_24 := BA_values[24];

    PLC_BA_DigOut_25 := BA_values[25];
    PLC_BA_DigOut_26 := BA_values[26];
    PLC_BA_DigOut_27 := BA_values[27];
    PLC_BA_DigOut_28 := BA_values[28];
    PLC_BA_DigOut_29 := BA_values[29];
    PLC_BA_DigOut_30 := BA_values[30];
    PLC_BA_DigOut_31 := BA_values[31];
    PLC_BA_DigOut_32 := BA_values[32];

END_FUNCTION

(* ---- BA_WriteConfigBits.st ---- *)
(****************************************************************************
**
** Copyright (C) 2021 Francesco Mandracci
** Contact: https://github.com/fmandracci/smart-home
**
** This file is part of the Smart Home Framework.
**
** Commercial License Usage
** Licensees holding valid commercial licenses may use this file in
** accordance with the terms contained in a written agreement
** between you and the copyright owner.
**
** GNU Lesser General Public License Usage
** Alternatively, this file may be used under the terms of the GNU Lesser
** General Public License version 3 as published by the Free Software
** Foundation and appearing in the file LICENSE included in the
** packaging of this file. Please review the following information to
** ensure the GNU Lesser General Public License version 3 requirements
** will be met: https://www.gnu.org/licenses/lgpl-3.0.html.
**
****************************************************************************)

FUNCTION BA_WriteConfigBits
#import "Crosstable.gvl"
#import "Resource1.gvl"
VAR_INPUT
    values: ARRAY [1..32] OF BOOL;
END_VAR;

        if PLC_control_type = ControlType_2 then
        (* MPNE_A, MPNE_B on RTU0 *)
            if MPNE_A_DigOut_17 <> values[ 1] then MPNE_A_DigOut_17 := values[ 1]; end_if;
            if MPNE_A_DigOut_18 <> values[ 2] then MPNE_A_DigOut_18 := values[ 2]; end_if;
            if MPNE_A_DigOut_19 <> values[ 3] then MPNE_A_DigOut_19 := values[ 3]; end_if;
            if MPNE_A_DigOut_20 <> values[ 4] then MPNE_A_DigOut_20 := values[ 4]; end_if;
            if MPNE_A_DigOut_21 <> values[ 5] then MPNE_A_DigOut_21 := values[ 5]; end_if;
            if MPNE_A_DigOut_22 <> values[ 6] then MPNE_A_DigOut_22 := values[ 6]; end_if;
            if MPNE_A_DigOut_23 <> values[ 7] then MPNE_A_DigOut_23 := values[ 7]; end_if;
            if MPNE_A_DigOut_24 <> values[ 8] then MPNE_A_DigOut_24 := values[ 8]; end_if;
            if MPNE_A_DigOut_25 <> values[ 9] then MPNE_A_DigOut_25 := values[ 9]; end_if;
            if MPNE_A_DigOut_26 <> values[10] then MPNE_A_DigOut_26 := values[10]; end_if;
            if MPNE_A_DigOut_27 <> values[11] then MPNE_A_DigOut_27 := values[11]; end_if;
            if MPNE_A_DigOut_28 <> values[12] then MPNE_A_DigOut_28 := values[12]; end_if;
            if MPNE_A_DigOut_29 <> values[13] then MPNE_A_DigOut_29 := values[13]; end_if;
            if MPNE_A_DigOut_30 <> values[14] then MPNE_A_DigOut_30 := values[14]; end_if;
            if MPNE_A_DigOut_31 <> values[15] then MPNE_A_DigOut_31 := values[15]; end_if;
            if MPNE_A_DigOut_32 <> values[16] then MPNE_A_DigOut_32 := values[16]; end_if;

            if MPNE_B_DigOut_17 <> values[17] then MPNE_B_DigOut_17 := values[17]; end_if;
            if MPNE_B_DigOut_18 <> values[18] then MPNE_B_DigOut_18 := values[18]; end_if;
            if MPNE_B_DigOut_19 <> values[19] then MPNE_B_DigOut_19 := values[19]; end_if;
            if MPNE_B_DigOut_20 <> values[20] then MPNE_B_DigOut_20 := values[20]; end_if;
            if MPNE_B_DigOut_21 <> values[21] then MPNE_B_DigOut_21 := values[21]; end_if;
            if MPNE_B_DigOut_22 <> values[22] then MPNE_B_DigOut_22 := values[22]; end_if;
            if MPNE_B_DigOut_23 <> values[23] then MPNE_B_DigOut_23 := values[23]; end_if;
            if MPNE_B_DigOut_24 <> values[24] then MPNE_B_DigOut_24 := values[24]; end_if;
            if MPNE_B_DigOut_25 <> values[25] then MPNE_B_DigOut_25 := values[25]; end_if;
            if MPNE_B_DigOut_26 <> values[26] then MPNE_B_DigOut_26 := values[26]; end_if;
            if MPNE_B_DigOut_27 <> values[27] then MPNE_B_DigOut_27 := values[27]; end_if;
            if MPNE_B_DigOut_28 <> values[28] then MPNE_B_DigOut_28 := values[28]; end_if;
            if MPNE_B_DigOut_29 <> values[29] then MPNE_B_DigOut_29 := values[29]; end_if;
            if MPNE_B_DigOut_30 <> values[30] then MPNE_B_DigOut_30 := values[30]; end_if;
            if MPNE_B_DigOut_31 <> values[31] then MPNE_B_DigOut_31 := values[31]; end_if;
            if MPNE_B_DigOut_32 <> values[32] then MPNE_B_DigOut_32 := values[32]; end_if;

        elsif PLC_control_type = ControlType_12 then
            (* Fast I/O on GPIO *)
            ; (* one enable only *)

        elsif PLC_control_type = ControlType_13 then
            (* TPAC1007_04_AD Local I/O on RTU3 *)
            ; (* one enable only *)

        elsif PLC_control_type = ControlType_6 then
            (* MPNC DI16 "A,B" + DO16 "A" on RTU0 *)
            if MPNC_DigOut_A_1  <> (values[ 1] or values[17]) then MPNC_DigOut_A_1  := (values[ 1] or values[17]); end_if;
            if MPNC_DigOut_A_2  <> (values[ 2] or values[18]) then MPNC_DigOut_A_2  := (values[ 2] or values[18]); end_if;
            if MPNC_DigOut_A_3  <> (values[ 3] or values[19]) then MPNC_DigOut_A_3  := (values[ 3] or values[19]); end_if;
            if MPNC_DigOut_A_4  <> (values[ 4] or values[20]) then MPNC_DigOut_A_4  := (values[ 4] or values[20]); end_if;
            if MPNC_DigOut_A_5  <> (values[ 5] or values[21]) then MPNC_DigOut_A_5  := (values[ 5] or values[21]); end_if;
            if MPNC_DigOut_A_6  <> (values[ 6] or values[22]) then MPNC_DigOut_A_6  := (values[ 6] or values[22]); end_if;
            if MPNC_DigOut_A_7  <> (values[ 7] or values[23]) then MPNC_DigOut_A_7  := (values[ 7] or values[23]); end_if;
            if MPNC_DigOut_A_8  <> (values[ 8] or values[24]) then MPNC_DigOut_A_8  := (values[ 8] or values[24]); end_if;
            if MPNC_DigOut_A_9  <> (values[ 9] or values[25]) then MPNC_DigOut_A_9  := (values[ 9] or values[25]); end_if;
            if MPNC_DigOut_A_10 <> (values[10] or values[26]) then MPNC_DigOut_A_10 := (values[10] or values[26]); end_if;
            if MPNC_DigOut_A_11 <> (values[11] or values[27]) then MPNC_DigOut_A_11 := (values[11] or values[27]); end_if;
            if MPNC_DigOut_A_12 <> (values[12] or values[28]) then MPNC_DigOut_A_12 := (values[12] or values[28]); end_if;
            if MPNC_DigOut_A_13 <> (values[13] or values[29]) then MPNC_DigOut_A_13 := (values[13] or values[29]); end_if;
            if MPNC_DigOut_A_14 <> (values[14] or values[30]) then MPNC_DigOut_A_14 := (values[14] or values[30]); end_if;
            if MPNC_DigOut_A_15 <> (values[15] or values[31]) then MPNC_DigOut_A_15 := (values[15] or values[31]); end_if;
            if MPNC_DigOut_A_16 <> (values[16] or values[32]) then MPNC_DigOut_A_16 := (values[16] or values[32]); end_if;

        elsif PLC_control_type = ControlType_14 then
            (* MPNC DI16 "A,B" + DO16 "A,B" on RTU0 *)
            if MPNC_DigOut_A_1  <> values[ 1] then MPNC_DigOut_A_1  := values[ 1]; end_if;
            if MPNC_DigOut_A_2  <> values[ 2] then MPNC_DigOut_A_2  := values[ 2]; end_if;
            if MPNC_DigOut_A_3  <> values[ 3] then MPNC_DigOut_A_3  := values[ 3]; end_if;
            if MPNC_DigOut_A_4  <> values[ 4] then MPNC_DigOut_A_4  := values[ 4]; end_if;
            if MPNC_DigOut_A_5  <> values[ 5] then MPNC_DigOut_A_5  := values[ 5]; end_if;
            if MPNC_DigOut_A_6  <> values[ 6] then MPNC_DigOut_A_6  := values[ 6]; end_if;
            if MPNC_DigOut_A_7  <> values[ 7] then MPNC_DigOut_A_7  := values[ 7]; end_if;
            if MPNC_DigOut_A_8  <> values[ 8] then MPNC_DigOut_A_8  := values[ 8]; end_if;
            if MPNC_DigOut_A_9  <> values[ 9] then MPNC_DigOut_A_9  := values[ 9]; end_if;
            if MPNC_DigOut_A_10 <> values[10] then MPNC_DigOut_A_10 := values[10]; end_if;
            if MPNC_DigOut_A_11 <> values[11] then MPNC_DigOut_A_11 := values[11]; end_if;
            if MPNC_DigOut_A_12 <> values[12] then MPNC_DigOut_A_12 := values[12]; end_if;
            if MPNC_DigOut_A_13 <> values[13] then MPNC_DigOut_A_13 := values[13]; end_if;
            if MPNC_DigOut_A_14 <> values[14] then MPNC_DigOut_A_14 := values[14]; end_if;
            if MPNC_DigOut_A_15 <> values[15] then MPNC_DigOut_A_15 := values[15]; end_if;
            if MPNC_DigOut_A_16 <> values[16] then MPNC_DigOut_A_16 := values[16]; end_if;

            if MPNC_DigOut_B_1  <> values[17] then MPNC_DigOut_B_1  := values[17]; end_if;
            if MPNC_DigOut_B_2  <> values[18] then MPNC_DigOut_B_2  := values[18]; end_if;
            if MPNC_DigOut_B_3  <> values[19] then MPNC_DigOut_B_3  := values[19]; end_if;
            if MPNC_DigOut_B_4  <> values[20] then MPNC_DigOut_B_4  := values[20]; end_if;
            if MPNC_DigOut_B_5  <> values[21] then MPNC_DigOut_B_5  := values[21]; end_if;
            if MPNC_DigOut_B_6  <> values[22] then MPNC_DigOut_B_6  := values[22]; end_if;
            if MPNC_DigOut_B_7  <> values[23] then MPNC_DigOut_B_7  := values[23]; end_if;
            if MPNC_DigOut_B_8  <> values[24] then MPNC_DigOut_B_8  := values[24]; end_if;
            if MPNC_DigOut_B_9  <> values[25] then MPNC_DigOut_B_9  := values[25]; end_if;
            if MPNC_DigOut_B_10 <> values[26] then MPNC_DigOut_B_10 := values[26]; end_if;
            if MPNC_DigOut_B_11 <> values[27] then MPNC_DigOut_B_11 := values[27]; end_if;
            if MPNC_DigOut_B_12 <> values[28] then MPNC_DigOut_B_12 := values[28]; end_if;
            if MPNC_DigOut_B_13 <> values[29] then MPNC_DigOut_B_13 := values[29]; end_if;
            if MPNC_DigOut_B_14 <> values[30] then MPNC_DigOut_B_14 := values[30]; end_if;
            if MPNC_DigOut_B_15 <> values[31] then MPNC_DigOut_B_15 := values[31]; end_if;
            if MPNC_DigOut_B_16 <> values[32] then MPNC_DigOut_B_16 := values[32]; end_if;

        end_if;

END_FUNCTION

(* ---- BA_WriteLeds.st ---- *)
(****************************************************************************
**
** Copyright (C) 2021 Francesco Mandracci
** Contact: https://github.com/fmandracci/smart-home
**
** This file is part of the Smart Home Framework.
**
** Commercial License Usage
** Licensees holding valid commercial licenses may use this file in
** accordance with the terms contained in a written agreement
** between you and the copyright owner.
**
** GNU Lesser General Public License Usage
** Alternatively, this file may be used under the terms of the GNU Lesser
** General Public License version 3 as published by the Free Software
** Foundation and appearing in the file LICENSE included in the
** packaging of this file. Please review the following information to
** ensure the GNU Lesser General Public License version 3 requirements
** will be met: https://www.gnu.org/licenses/lgpl-3.0.html.
**
****************************************************************************)

FUNCTION BA_WriteLeds
#import "Crosstable.gvl"
#import "Resource1.gvl"
VAR_INPUT
    index : UINT;
    status : UINT;
END_VAR
VAR
	green    : BOOL;
	red      : BOOL;
	yellow1  : BOOL;
	yellow2  : BOOL;

	siren    : BOOL;
	enable_A : BOOL;
	enable_B : BOOL;
	enable_C : BOOL;
END_VAR;

	(* ----- checking ----- *)

	case status of

	ALARM_STATUS_ZERO:
		green    := false;
		red      := false;
		yellow1  := false;
		yellow2  := false;

		siren    := false;
		enable_A := false;
		enable_B := false;
		enable_C := false;

	ALARM_STATUS_OFF:
		green    := false;
		red      := false;
		yellow1  := false;
		yellow2  := false;

		siren    := false;
		enable_A := false;
		enable_B := false;
		enable_C := false;

	ALARM_STATUS_ARMED:
		green    := (PLC_Seconds mod 2) = 0; (* blinking 1 s on and 1 s off *)
		red      := false;
		yellow1  := (index = ALARM_INDEX_NIGHTTIME) or (index = ALARM_INDEX_EVERYTHING);
		yellow2  := (index = ALARM_INDEX_DAYTIME) or (index = ALARM_INDEX_EVERYTHING);

		siren    := false;
		enable_A := (index = ALARM_INDEX_DAYTIME) or (index = ALARM_INDEX_NIGHTTIME) or (index = ALARM_INDEX_EVERYTHING);
		enable_B := (index = ALARM_INDEX_NIGHTTIME) or (index = ALARM_INDEX_EVERYTHING);
		enable_C := (index = ALARM_INDEX_EVERYTHING);

	ALARM_STATUS_ENABLED:
		green    := true;
		red      := false;
		yellow1  := (index = ALARM_INDEX_NIGHTTIME) or (index = ALARM_INDEX_EVERYTHING);
		yellow2  := (index = ALARM_INDEX_DAYTIME) or (index = ALARM_INDEX_EVERYTHING);

		siren    := false;
		enable_A := (index = ALARM_INDEX_DAYTIME) or (index = ALARM_INDEX_NIGHTTIME) or (index = ALARM_INDEX_EVERYTHING);
		enable_B := (index = ALARM_INDEX_NIGHTTIME) or (index = ALARM_INDEX_EVERYTHING);
		enable_C := (index = ALARM_INDEX_EVERYTHING);

	ALARM_STATUS_RINGING:
		green    := true;
		red      := (PLC_Seconds mod 2) = 0; (* blinking 1 s on and 1 s off *)
		yellow1  := (index = ALARM_INDEX_NIGHTTIME) or (index = ALARM_INDEX_EVERYTHING);
		yellow2  := (index = ALARM_INDEX_DAYTIME) or (index = ALARM_INDEX_EVERYTHING);

		siren    := true; (********************** SIREN *******************************)
		enable_A := (index = ALARM_INDEX_DAYTIME) or (index = ALARM_INDEX_NIGHTTIME) or (index = ALARM_INDEX_EVERYTHING);
		enable_B := (index = ALARM_INDEX_NIGHTTIME) or (index = ALARM_INDEX_EVERYTHING);
		enable_C := (index = ALARM_INDEX_EVERYTHING);

	ALARM_STATUS_MUTED:
		green    := true;
		red      := true;
		yellow1  := (index = ALARM_INDEX_NIGHTTIME) or (index = ALARM_INDEX_EVERYTHING);
		yellow2  := (index = ALARM_INDEX_DAYTIME) or (index = ALARM_INDEX_EVERYTHING);

		siren    := false;
		enable_A := (index = ALARM_INDEX_DAYTIME) or (index = ALARM_INDEX_NIGHTTIME) or (index = ALARM_INDEX_EVERYTHING);
		enable_B := (index = ALARM_INDEX_NIGHTTIME) or (index = ALARM_INDEX_EVERYTHING);
		enable_C := (index = ALARM_INDEX_EVERYTHING);

	ALARM_STATUS_TESTING:
		(* values from page046 *)
		green    := PLC_BA_led_green;
		red      := PLC_BA_led_red;
		yellow1  := PLC_BA_led_yellow1;
		yellow2  := PLC_BA_led_yellow2;

		siren    := PLC_BA_siren;
		enable_A := PLC_BA_relay_A;
		enable_B := PLC_BA_relay_B;
		enable_C := PLC_BA_relay_C;

	else
		green    := false;
		red      := false;
		yellow1  := false;
		yellow2  := false;

		siren    := false;
		enable_A := false;
		enable_B := false;
		enable_C := false;

	end_case;

	(* ----- crosstable assignments -----*)

    PLC_BA_led_green   := green       ;
    PLC_BA_led_red     := red         ;
    PLC_BA_led_yellow1 := yellow1     ;
    PLC_BA_led_yellow2 := yellow2     ;

    if SRV_BA_led_green   <> green   then SRV_BA_led_green   := green  ; end_if;
    if SRV_BA_led_red     <> red     then SRV_BA_led_red     := red    ; end_if;
    if SRV_BA_led_yellow1 <> yellow1 then SRV_BA_led_yellow1 := yellow1; end_if;
    if SRV_BA_led_yellow2 <> yellow2 then SRV_BA_led_yellow2 := yellow2; end_if;

    PLC_BA_siren       := siren       ;
    PLC_BA_relay_A     := enable_A    ;
    PLC_BA_relay_B     := enable_B    ;
    PLC_BA_relay_C     := enable_C    ;

	(* ----- fieldbus assignments ----- *)

    BA_SetDigOuts(green, red, yellow1, yellow2, siren, enable_A, enable_B, enable_C);

END_FUNCTION

(* ---- EP_ManageRequest.st ---- *)
(****************************************************************************
**
** Copyright (C) 2021 Francesco Mandracci
** Contact: https://github.com/fmandracci/smart-home
**
** This file is part of the Smart Home Framework.
**
** Commercial License Usage
** Licensees holding valid commercial licenses may use this file in
** accordance with the terms contained in a written agreement
** between you and the copyright owner.
**
** GNU Lesser General Public License Usage
** Alternatively, this file may be used under the terms of the GNU Lesser
** General Public License version 3 as published by the Free Software
** Foundation and appearing in the file LICENSE included in the
** packaging of this file. Please review the following information to
** ensure the GNU Lesser General Public License version 3 requirements
** will be met: https://www.gnu.org/licenses/lgpl-3.0.html.
**
****************************************************************************)

FUNCTION EP_ManageRequest
#import "Crosstable.gvl"
#import "Resource1.gvl"
VAR_INPUT
	n : UINT;
	Tn_requested_W: UINT;
END_VAR
VAR_IN_OUT
	Tn_assigned_W: UINT;
	total_requested_W: UINT;
	total_assigned_W: UINT;
	last_assigned: UINT;
	first_refused: UINT;
END_VAR

	total_requested_W := total_requested_W + Tn_requested_W;

	if n > PLC_Tn_count or Tn_requested_W = 0 or PLC_EP_BlackoutDetected or PLC_EP_OverloadDetected then
		Tn_assigned_W := 0;

	elsif (total_assigned_W + Tn_requested_W) <= PLC_EP_max_assigned_W and (total_assigned_W + Tn_requested_W) <= PLC_EP_overload_W then
		Tn_assigned_W := Tn_requested_W;
		total_assigned_W := total_assigned_W + Tn_requested_W;
		last_assigned := n;

	else
		Tn_assigned_W := 0;
		if first_refused = 0 then
			first_refused := n;
		end_if;

	end_if;

END_FUNCTION

(* ---- EP_SetDigOut_relay.st ---- *)
(****************************************************************************
**
** Copyright (C) 2021 Francesco Mandracci
** Contact: https://github.com/fmandracci/smart-home
**
** This file is part of the Smart Home Framework.
**
** Commercial License Usage
** Licensees holding valid commercial licenses may use this file in
** accordance with the terms contained in a written agreement
** between you and the copyright owner.
**
** GNU Lesser General Public License Usage
** Alternatively, this file may be used under the terms of the GNU Lesser
** General Public License version 3 as published by the Free Software
** Foundation and appearing in the file LICENSE included in the
** packaging of this file. Please review the following information to
** ensure the GNU Lesser General Public License version 3 requirements
** will be met: https://www.gnu.org/licenses/lgpl-3.0.html.
**
****************************************************************************)

FUNCTION EP_SetDigOut_relay
#import "Crosstable.gvl"
#import "Resource1.gvl"
VAR_INPUT
    n : UINT;
    value : BOOL;
END_VAR

	if PLC_control_type = ControlType_1 then
		if PLC_PRODUCT_ID = 16#1043030C then
			(* Fast I/O on GPIO *);
			case n of
        	1: if PLC_FastIO_5 <> value then PLC_FastIO_5 := value; end_if;
        	2: if PLC_FastIO_6 <> value then PLC_FastIO_6 := value; end_if;
        	3: if PLC_FastIO_7 <> value then PLC_FastIO_7 := value; end_if;
        	4: if PLC_FastIO_8 <> value then PLC_FastIO_8 := value; end_if;
			else ;
			end_case;
		elsif PLC_PRODUCT_ID = 16#100704AD or PLC_PRODUCT_ID = 16#100704AE or PLC_PRODUCT_ID = 16#100704AA or PLC_PRODUCT_ID = 16#100704AC then
			case n of
        	1: if PLC_DigDir_1 <> DigDir_OUT then PLC_DigDir_1 := DigDir_OUT; end_if;
        	2: if PLC_DigDir_2 <> DigDir_OUT then PLC_DigDir_2 := DigDir_OUT; end_if;
        	3: if PLC_DigDir_3 <> DigDir_OUT then PLC_DigDir_3 := DigDir_OUT; end_if;
        	4: if PLC_DigDir_4 <> DigDir_OUT then PLC_DigDir_4 := DigDir_OUT; end_if;
        	5: if PLC_DigDir_5 <> DigDir_OUT then PLC_DigDir_5 := DigDir_OUT; end_if;
        	6: if PLC_DigDir_6 <> DigDir_OUT then PLC_DigDir_6 := DigDir_OUT; end_if;
        	7: if PLC_DigDir_7 <> DigDir_OUT then PLC_DigDir_7 := DigDir_OUT; end_if;
        	8: if PLC_DigDir_8 <> DigDir_OUT then PLC_DigDir_8 := DigDir_OUT; end_if;
			else ;
			end_case;
			case n of
        	1: if PLC_DigOut_1 <> value then PLC_DigOut_1 := value; end_if;
        	2: if PLC_DigOut_2 <> value then PLC_DigOut_2 := value; end_if;
        	3: if PLC_DigOut_3 <> value then PLC_DigOut_3 := value; end_if;
        	4: if PLC_DigOut_4 <> value then PLC_DigOut_4 := value; end_if;
        	5: if PLC_DigOut_5 <> value then PLC_DigOut_5 := value; end_if;
        	6: if PLC_DigOut_6 <> value then PLC_DigOut_6 := value; end_if;
        	7: if PLC_DigOut_7 <> value then PLC_DigOut_7 := value; end_if;
        	8: if PLC_DigOut_8 <> value then PLC_DigOut_8 := value; end_if;
			else ;
			end_case;
		else
			; (* TP.. *)
		end_if;

	elsif PLC_control_type = ControlType_7 then
		(* Fast I/O 7,8 on GPIO *);
		case n of
    	1: if PLC_FastIO_7 <> value then PLC_FastIO_7 := value; end_if;
    	2: if PLC_FastIO_8 <> value then PLC_FastIO_8 := value; end_if;
		else ;
		end_case;

	elsif PLC_control_type = ControlType_12 then
		(* Fast I/O on GPIO *);
		case n of
    	1: if PLC_FastIO_7 <> value then PLC_FastIO_7 := value; end_if;
		else ;
		end_case;

	elsif PLC_control_type = ControlType_13 then
		(* TPAC1007_04_AD Local I/O on RTU3 *)
		case n of
    	1: if PLC_DigDir_7 <> DigDir_OUT then PLC_DigDir_7 := DigDir_OUT; end_if;
    	2: if PLC_DigDir_8 <> DigDir_OUT then PLC_DigDir_8 := DigDir_OUT; end_if;
		else ;
		end_case;
		case n of
    	1: if PLC_DigOut_7 <> value then PLC_DigOut_7 := value; end_if;
    	2: if PLC_DigOut_8 <> value then PLC_DigOut_8 := value; end_if;
		else ;
		end_case;

	elsif PLC_control_type = ControlType_6 then
		(* n=1..4: MPNC base DigOut_1..4 *)
		case n of
		1:
	    	if MPNC_DigDir_1 <> DigDir_OUT then MPNC_DigDir_1 := DigDir_OUT; end_if;
	        if MPNC_DigOut_1 <> value      then MPNC_DigOut_1 := value     ; end_if;
		2:
	    	if MPNC_DigDir_2 <> DigDir_OUT then MPNC_DigDir_2 := DigDir_OUT; end_if;
	        if MPNC_DigOut_2 <> value      then MPNC_DigOut_2 := value     ; end_if;
		3:
	    	if MPNC_DigDir_3 <> DigDir_OUT then MPNC_DigDir_3 := DigDir_OUT; end_if;
	        if MPNC_DigOut_3 <> value      then MPNC_DigOut_3 := value     ; end_if;
		4:
	    	if MPNC_DigDir_4 <> DigDir_OUT then MPNC_DigDir_4 := DigDir_OUT; end_if;
	        if MPNC_DigOut_4 <> value      then MPNC_DigOut_4 := value     ; end_if;
		else ;
		end_case;

	elsif PLC_control_type = ControlType_14 then
		(* MPNC DO16 "C" on RTU0 *)
		case n of
    	1: if MPNC_DigOut_C_1 <> value then MPNC_DigOut_C_1 := value; end_if;
    	2: if MPNC_DigOut_C_2 <> value then MPNC_DigOut_C_2 := value; end_if;
    	3: if MPNC_DigOut_C_3 <> value then MPNC_DigOut_C_3 := value; end_if;
    	4: if MPNC_DigOut_C_4 <> value then MPNC_DigOut_C_4 := value; end_if;
    	5: if MPNC_DigOut_C_5 <> value then MPNC_DigOut_C_5 := value; end_if;
    	6: if MPNC_DigOut_C_6 <> value then MPNC_DigOut_C_6 := value; end_if;
    	7: if MPNC_DigOut_C_7 <> value then MPNC_DigOut_C_7 := value; end_if;
    	8: if MPNC_DigOut_C_8 <> value then MPNC_DigOut_C_8 := value; end_if;
		else ;
		end_case;

	elsif PLC_control_type = ControlType_15 then

		case n of
    	1: if PLC_DigDir_1 <> DigDir_OUT then PLC_DigDir_1 := DigDir_OUT; end_if;
    	2: if PLC_DigDir_2 <> DigDir_OUT then PLC_DigDir_2 := DigDir_OUT; end_if;
    	3: if PLC_DigDir_3 <> DigDir_OUT then PLC_DigDir_3 := DigDir_OUT; end_if;
    	4: if PLC_DigDir_4 <> DigDir_OUT then PLC_DigDir_4 := DigDir_OUT; end_if;
    	5: if PLC_DigDir_5 <> DigDir_OUT then PLC_DigDir_5 := DigDir_OUT; end_if;
    	6: if PLC_DigDir_6 <> DigDir_OUT then PLC_DigDir_6 := DigDir_OUT; end_if;
    	7: if PLC_DigDir_7 <> DigDir_OUT then PLC_DigDir_7 := DigDir_OUT; end_if;
		else ;
		end_case;
		case n of
    	1: if PLC_DigOut_1 <> value then PLC_DigOut_1 := value; end_if;
    	2: if PLC_DigOut_2 <> value then PLC_DigOut_2 := value; end_if;
    	3: if PLC_DigOut_3 <> value then PLC_DigOut_3 := value; end_if;
    	4: if PLC_DigOut_4 <> value then PLC_DigOut_4 := value; end_if;
    	5: if PLC_DigOut_5 <> value then PLC_DigOut_5 := value; end_if;
    	6: if PLC_DigOut_6 <> value then PLC_DigOut_6 := value; end_if;
    	7: if PLC_DigOut_7 <> value then PLC_DigOut_7 := value; end_if;
		else ;
		end_case;

	end_if;

END_FUNCTION

(* ---- EP_Wattmeter.st ---- *)
(****************************************************************************
**
** Copyright (C) 2021 Francesco Mandracci
** Contact: https://github.com/fmandracci/smart-home
**
** This file is part of the Smart Home Framework.
**
** Commercial License Usage
** Licensees holding valid commercial licenses may use this file in
** accordance with the terms contained in a written agreement
** between you and the copyright owner.
**
** GNU Lesser General Public License Usage
** Alternatively, this file may be used under the terms of the GNU Lesser
** General Public License version 3 as published by the Free Software
** Foundation and appearing in the file LICENSE included in the
** packaging of this file. Please review the following information to
** ensure the GNU Lesser General Public License version 3 requirements
** will be met: https://www.gnu.org/licenses/lgpl-3.0.html.
**
****************************************************************************)

FUNCTION EP_Wattmeter
#import "Crosstable.gvl"
#import "Resource1.gvl"
VAR_INPUT
	n : UINT;
END_VAR
VAR_IN_OUT
	W    : INT;   (*  W  *)
	_var : INT;   (* var *)
	VA   : INT;   (* VA  *)
	kWh  : DINT;  (* kWh *)
END_VAR

	if PLC_control_type <> ControlType_6 then

		case n of
		 1:
		 	W   := REAL_TO_INT  (RTU_EP_wattmeter_M_P             );
			_var:= REAL_TO_INT  (RTU_EP_wattmeter_M_Q             );
			VA  := REAL_TO_INT  (RTU_EP_wattmeter_M_S             );
			kWh := REAL_TO_DINT (RTU_EP_wattmeter_M_Ein  /  100.0) + PLC_EP_wattmeter_M_kWh_offset; (* wxyz Wh --> w.x kWh *)
		 2:
		 	W   := REAL_TO_INT  (RTU_EP_wattmeter_F_P             );
			_var:= REAL_TO_INT  (RTU_EP_wattmeter_F_Q             );
			VA  := REAL_TO_INT  (RTU_EP_wattmeter_F_S             );
			kWh := REAL_TO_DINT (RTU_EP_wattmeter_F_Ein  /  100.0) + PLC_EP_wattmeter_F_kWh_offset; (* wxyz Wh --> w.x kWh *)
		 3:
		 	W   := REAL_TO_INT  (RTU_EP_wattmeter01_P             );
			_var:= REAL_TO_INT  (RTU_EP_wattmeter01_Q             );
			VA  := REAL_TO_INT  (RTU_EP_wattmeter01_S             );
			kWh := REAL_TO_DINT (RTU_EP_wattmeter01_Ein  /  100.0) + PLC_EP_wattmeter01_kWh_offset; (* wxyz Wh --> w.x kWh *)
		 4:
		 	W   := REAL_TO_INT  (RTU_EP_wattmeter02_P             );
			_var:= REAL_TO_INT  (RTU_EP_wattmeter02_Q             );
			VA  := REAL_TO_INT  (RTU_EP_wattmeter02_S             );
			kWh := REAL_TO_DINT (RTU_EP_wattmeter02_Ein  /  100.0) + PLC_EP_wattmeter02_kWh_offset; (* wxyz Wh --> w.x kWh *)
		 5:
		 	W   := REAL_TO_INT  (RTU_EP_wattmeter03_P             );
			_var:= REAL_TO_INT  (RTU_EP_wattmeter03_Q             );
			VA  := REAL_TO_INT  (RTU_EP_wattmeter03_S             );
			kWh := REAL_TO_DINT (RTU_EP_wattmeter03_Ein  /  100.0) + PLC_EP_wattmeter03_kWh_offset; (* wxyz Wh --> w.x kWh *)
		 6:
		 	W   := REAL_TO_INT  (RTU_EP_wattmeter04_P             );
			_var:= REAL_TO_INT  (RTU_EP_wattmeter04_Q             );
			VA  := REAL_TO_INT  (RTU_EP_wattmeter04_S             );
			kWh := REAL_TO_DINT (RTU_EP_wattmeter04_Ein  /  100.0) + PLC_EP_wattmeter04_kWh_offset; (* wxyz Wh --> w.x kWh *)
		 7:
		 	W   := REAL_TO_INT  (RTU_EP_wattmeter05_P             );
			_var:= REAL_TO_INT  (RTU_EP_wattmeter05_Q             );
			VA  := REAL_TO_INT  (RTU_EP_wattmeter05_S             );
			kWh := REAL_TO_DINT (RTU_EP_wattmeter05_Ein  /  100.0) + PLC_EP_wattmeter05_kWh_offset; (* wxyz Wh --> w.x kWh *)
		 8:
		 	W   := REAL_TO_INT  (RTU_EP_wattmeter06_P             );
			_var:= REAL_TO_INT  (RTU_EP_wattmeter06_Q             );
			VA  := REAL_TO_INT  (RTU_EP_wattmeter06_S             );
			kWh := REAL_TO_DINT (RTU_EP_wattmeter06_Ein  /  100.0) + PLC_EP_wattmeter06_kWh_offset; (* wxyz Wh --> w.x kWh *)
		 9:
		 	W   := REAL_TO_INT  (RTU_EP_wattmeter07_P             );
			_var:= REAL_TO_INT  (RTU_EP_wattmeter07_Q             );
			VA  := REAL_TO_INT  (RTU_EP_wattmeter07_S             );
			kWh := REAL_TO_DINT (RTU_EP_wattmeter07_Ein  /  100.0) + PLC_EP_wattmeter07_kWh_offset; (* wxyz Wh --> w.x kWh *)
		10:
		 	W   := REAL_TO_INT  (RTU_EP_wattmeter08_P             );
			_var:= REAL_TO_INT  (RTU_EP_wattmeter08_Q             );
			VA  := REAL_TO_INT  (RTU_EP_wattmeter08_S             );
			kWh := REAL_TO_DINT (RTU_EP_wattmeter08_Ein  /  100.0) + PLC_EP_wattmeter08_kWh_offset; (* wxyz Wh --> w.x kWh *)
		11:
		 	W   := REAL_TO_INT  (RTU_EP_wattmeter09_P             );
			_var:= REAL_TO_INT  (RTU_EP_wattmeter09_Q             );
			VA  := REAL_TO_INT  (RTU_EP_wattmeter09_S             );
			kWh := REAL_TO_DINT (RTU_EP_wattmeter09_Ein  /  100.0) + PLC_EP_wattmeter09_kWh_offset; (* wxyz Wh --> w.x kWh *)
		12:
		 	W   := REAL_TO_INT  (RTU_EP_wattmeter10_P             );
			_var:= REAL_TO_INT  (RTU_EP_wattmeter10_Q             );
			VA  := REAL_TO_INT  (RTU_EP_wattmeter10_S             );
			kWh := REAL_TO_DINT (RTU_EP_wattmeter10_Ein  /  100.0) + PLC_EP_wattmeter10_kWh_offset; (* wxyz Wh --> w.x kWh *)
		else ;
		end_case;

    elsif PLC_control_type = ControlType_6 then

		case n of
		 1:
		 	W   := REAL_TO_INT  (SysActivePower_0             );
			_var:= REAL_TO_INT  (SysReactivePower_0           );
			VA  := REAL_TO_INT  (SysApparentPower_0           );
			kWh := REAL_TO_DINT (SysImpActiveEnergy_0  / 100.0) + PLC_EP_wattmeter_M_kWh_offset; (* wxyz Wh --> w.x kWh *)
		 2:
		 	W   := REAL_TO_INT  (SysActivePower_1             );
			_var:= REAL_TO_INT  (SysReactivePower_1           );
			VA  := REAL_TO_INT  (SysApparentPower_1           );
			kWh := REAL_TO_DINT (SysImpActiveEnergy_1  / 100.0) + PLC_EP_wattmeter_F_kWh_offset; (* wxyz Wh --> w.x kWh *)
		 3:
		 	W   := REAL_TO_INT  (SysActivePower_2             );
			_var:= REAL_TO_INT  (SysReactivePower_2           );
			VA  := REAL_TO_INT  (SysApparentPower_2           );
			kWh := REAL_TO_DINT (SysImpActiveEnergy_2  / 100.0) + PLC_EP_wattmeter01_kWh_offset; (* wxyz Wh --> w.x kWh *)
		 4:
		 	W   := REAL_TO_INT  (SysActivePower_3             );
			_var:= REAL_TO_INT  (SysReactivePower_3           );
			VA  := REAL_TO_INT  (SysApparentPower_3           );
			kWh := REAL_TO_DINT (SysImpActiveEnergy_3  / 100.0) + PLC_EP_wattmeter02_kWh_offset; (* wxyz Wh --> w.x kWh *)
		 5:
		 	W   := REAL_TO_INT  (SysActivePower_4             );
			_var:= REAL_TO_INT  (SysReactivePower_4           );
			VA  := REAL_TO_INT  (SysApparentPower_4           );
			kWh := REAL_TO_DINT (SysImpActiveEnergy_4  / 100.0) + PLC_EP_wattmeter03_kWh_offset; (* wxyz Wh --> w.x kWh *)
		 6:
		 	W   := REAL_TO_INT  (SysActivePower_5             );
			_var:= REAL_TO_INT  (SysReactivePower_5           );
			VA  := REAL_TO_INT  (SysApparentPower_5           );
			kWh := REAL_TO_DINT (SysImpActiveEnergy_5  / 100.0) + PLC_EP_wattmeter04_kWh_offset; (* wxyz Wh --> w.x kWh *)
		 7:
		 	W   := REAL_TO_INT  (SysActivePower_6             );
			_var:= REAL_TO_INT  (SysReactivePower_6           );
			VA  := REAL_TO_INT  (SysApparentPower_6           );
			kWh := REAL_TO_DINT (SysImpActiveEnergy_6  / 100.0) + PLC_EP_wattmeter05_kWh_offset; (* wxyz Wh --> w.x kWh *)
		 8:
		 	W   := REAL_TO_INT  (SysActivePower_7             );
			_var:= REAL_TO_INT  (SysReactivePower_7           );
			VA  := REAL_TO_INT  (SysApparentPower_7           );
			kWh := REAL_TO_DINT (SysImpActiveEnergy_7  / 100.0) + PLC_EP_wattmeter06_kWh_offset; (* wxyz Wh --> w.x kWh *)
		 9:
		 	W   := REAL_TO_INT  (SysActivePower_8             );
			_var:= REAL_TO_INT  (SysReactivePower_8           );
			VA  := REAL_TO_INT  (SysApparentPower_8           );
			kWh := REAL_TO_DINT (SysImpActiveEnergy_8  / 100.0) + PLC_EP_wattmeter07_kWh_offset; (* wxyz Wh --> w.x kWh *)
		10:
		 	W   := REAL_TO_INT  (SysActivePower_9             );
			_var:= REAL_TO_INT  (SysReactivePower_9           );
			VA  := REAL_TO_INT  (SysApparentPower_9           );
			kWh := REAL_TO_DINT (SysImpActiveEnergy_9  / 100.0) + PLC_EP_wattmeter08_kWh_offset; (* wxyz Wh --> w.x kWh *)
		11:
		 	W   := REAL_TO_INT  (SysActivePower_10            );
			_var:= REAL_TO_INT  (SysReactivePower_10          );
			VA  := REAL_TO_INT  (SysApparentPower_10          );
			kWh := REAL_TO_DINT (SysImpActiveEnergy_10 / 100.0) + PLC_EP_wattmeter09_kWh_offset; (* wxyz Wh --> w.x kWh *)
		12:
		 	W   := REAL_TO_INT  (SysActivePower_11            );
			_var:= REAL_TO_INT  (SysReactivePower_11          );
			VA  := REAL_TO_INT  (SysApparentPower_11          );
			kWh := REAL_TO_DINT (SysImpActiveEnergy_11 / 100.0) + PLC_EP_wattmeter10_kWh_offset; (* wxyz Wh --> w.x kWh *)
		else ;
		end_case;

	end_if;

END_FUNCTION

(* ---- EP_WattmeterFull.st ---- *)
(****************************************************************************
**
** Copyright (C) 2021 Francesco Mandracci
** Contact: https://github.com/fmandracci/smart-home
**
** This file is part of the Smart Home Framework.
**
** Commercial License Usage
** Licensees holding valid commercial licenses may use this file in
** accordance with the terms contained in a written agreement
** between you and the copyright owner.
**
** GNU Lesser General Public License Usage
** Alternatively, this file may be used under the terms of the GNU Lesser
** General Public License version 3 as published by the Free Software
** Foundation and appearing in the file LICENSE included in the
** packaging of this file. Please review the following information to
** ensure the GNU Lesser General Public License version 3 requirements
** will be met: https://www.gnu.org/licenses/lgpl-3.0.html.
**
****************************************************************************)

FUNCTION EP_WattmeterFull
#import "Crosstable.gvl"
#import "Resource1.gvl"
VAR_INPUT
	n : UINT;
END_VAR
VAR_IN_OUT
	W     : INT;   (*  W  *)
	_var  : INT;   (* var *)
	VA    : INT;   (* VA  *)
	pf    : INT;   (*  .  *)
	Hz    : INT;   (*  Hz *)
	V     : INT;   (*  V  *)
	A1    : INT;   (*  A  *)
	A2    : INT;   (*  A  *)
	A3    : INT;   (*  A  *)
	A     : INT;   (*  A  *)
	kWh   : DINT;  (* kWh *)
	e_kWh : DINT;  (* kWh *)
END_VAR

    if PLC_control_type <> ControlType_6 then

        case n of
        1:
            EP_Wattmeter(n, W, _var, VA, kWh);
            pf    := REAL_TO_INT  (RTU_EP_wattmeter_M_C  * 1000.0);
            Hz    := REAL_TO_INT  (RTU_EP_wattmeter_M_F  *  100.0);
            V     := REAL_TO_INT  (RTU_EP_wattmeter_M_U  *  100.0);
            A1    := REAL_TO_INT  (RTU_EP_wattmeter_M_I1 * 1000.0);
            A2    := REAL_TO_INT  (RTU_EP_wattmeter_M_I2 * 1000.0);
            A3    := REAL_TO_INT  (RTU_EP_wattmeter_M_I3 * 1000.0);
            A     := REAL_TO_INT  (RTU_EP_wattmeter_M_I  * 1000.0);
            e_kWh := REAL_TO_DINT (RTU_EP_wattmeter_M_Eout /  100.0) + PLC_EP_wattmeter_M_e_kWh_offset; (* wxyz Wh --> w.x kWh *)
        2:
            EP_Wattmeter(n, W, _var, VA, kWh);
            pf    := REAL_TO_INT  (RTU_EP_wattmeter_F_C  * 1000.0);
            Hz    := REAL_TO_INT  (RTU_EP_wattmeter_F_F  *  100.0);
            V     := REAL_TO_INT  (RTU_EP_wattmeter_F_U  *  100.0);
            A1    := REAL_TO_INT  (RTU_EP_wattmeter_F_I1 * 1000.0);
            A2    := REAL_TO_INT  (RTU_EP_wattmeter_F_I2 * 1000.0);
            A3    := REAL_TO_INT  (RTU_EP_wattmeter_F_I3 * 1000.0);
            A     := REAL_TO_INT  (RTU_EP_wattmeter_F_I  * 1000.0);
            e_kWh := REAL_TO_DINT (RTU_EP_wattmeter_F_Eout /  100.0) + PLC_EP_wattmeter_F_e_kWh_offset; (* wxyz Wh --> w.x kWh *)
        else ;
        end_case;

    elsif PLC_control_type = ControlType_6 then

        case n of
        1:
            EP_Wattmeter(n, W, _var, VA, kWh);
            pf    := REAL_TO_INT  (SysPowerFactor_0     * 1000.0);
            Hz    := REAL_TO_INT  (Frequency_0          *  100.0);
            V     := REAL_TO_INT  (SystemVoltage_0      *  100.0);
            A     := REAL_TO_INT  (SystemCurrent_0      * 1000.0);
            e_kWh := REAL_TO_DINT(SysExpActiveEnergy_0 /  100.0) + PLC_EP_wattmeter_M_e_kWh_offset; (* wxyz Wh --> w.x kWh *)
        2:
            EP_Wattmeter(n, W, _var, VA, kWh);
            pf    := REAL_TO_INT  (SysPowerFactor_1     * 1000.0);
         (* Hz    := REAL_TO_INT  (Frequency_1          *  100.0); *)
         (* V     := REAL_TO_INT  (SystemVoltage_1      *  100.0); *)
         (* A     := REAL_TO_INT  (SystemCurrent_1      * 1000.0); *)
            e_kWh := REAL_TO_DINT (SysExpActiveEnergy_1 /  100.0) + PLC_EP_wattmeter_F_e_kWh_offset; (* wxyz Wh --> w.x kWh *)
        else ;
        end_case;

    end_if;

END_FUNCTION

(* ---- getBit.st ---- *)
(****************************************************************************
**
** Copyright (C) 2021 Francesco Mandracci
** Contact: https://github.com/fmandracci/smart-home
**
** This file is part of the Smart Home Framework.
**
** Commercial License Usage
** Licensees holding valid commercial licenses may use this file in
** accordance with the terms contained in a written agreement
** between you and the copyright owner.
**
** GNU Lesser General Public License Usage
** Alternatively, this file may be used under the terms of the GNU Lesser
** General Public License version 3 as published by the Free Software
** Foundation and appearing in the file LICENSE included in the
** packaging of this file. Please review the following information to
** ensure the GNU Lesser General Public License version 3 requirements
** will be met: https://www.gnu.org/licenses/lgpl-3.0.html.
**
****************************************************************************)

FUNCTION getBit : BOOL
VAR_INPUT
    u : UINT;
    mask : WORD;
END_VAR
VAR
	w : WORD;
END_VAR

	w := UINT_TO_WORD(u);
	getBit := (w and mask) <> 0;

END_FUNCTION

(* ---- SetAnIn_PT100R.st ---- *)
(****************************************************************************
**
** Copyright (C) 2021 Francesco Mandracci
** Contact: https://github.com/fmandracci/smart-home
**
** This file is part of the Smart Home Framework.
**
** Commercial License Usage
** Licensees holding valid commercial licenses may use this file in
** accordance with the terms contained in a written agreement
** between you and the copyright owner.
**
** GNU Lesser General Public License Usage
** Alternatively, this file may be used under the terms of the GNU Lesser
** General Public License version 3 as published by the Free Software
** Foundation and appearing in the file LICENSE included in the
** packaging of this file. Please review the following information to
** ensure the GNU Lesser General Public License version 3 requirements
** will be met: https://www.gnu.org/licenses/lgpl-3.0.html.
**
****************************************************************************)

FUNCTION SetAnIn_PT100R
VAR_IN_OUT
	AnInConf_N : UINT;
	AnInNFilter : UINT;
END_VAR
	if AnInConf_N <> AnIn_PT100R then
		AnInConf_N := AnIn_PT100R;
	end_if;
	if AnInNFilter <> AnIn_LowPass then
		AnInNFilter := AnIn_LowPass;
	end_if;
END_FUNCTION

(* ---- setBit.st ---- *)
(****************************************************************************
**
** Copyright (C) 2021 Francesco Mandracci
** Contact: https://github.com/fmandracci/smart-home
**
** This file is part of the Smart Home Framework.
**
** Commercial License Usage
** Licensees holding valid commercial licenses may use this file in
** accordance with the terms contained in a written agreement
** between you and the copyright owner.
**
** GNU Lesser General Public License Usage
** Alternatively, this file may be used under the terms of the GNU Lesser
** General Public License version 3 as published by the Free Software
** Foundation and appearing in the file LICENSE included in the
** packaging of this file. Please review the following information to
** ensure the GNU Lesser General Public License version 3 requirements
** will be met: https://www.gnu.org/licenses/lgpl-3.0.html.
**
****************************************************************************)

FUNCTION setBit
VAR_INPUT
    mask : WORD;
    value : BOOL;
END_VAR
VAR_IN_OUT
    u : UINT;
END_VAR
VAR
	w : WORD;
END_VAR

	w := UINT_TO_WORD(u);
	if value then
		w := w or mask;
	else
		w := w and not mask;
	end_if;
	u := WORD_TO_UINT(w);

END_FUNCTION

(* ---- SetMpneDigDir_IN.st ---- *)
(****************************************************************************
**
** Copyright (C) 2021 Francesco Mandracci
** Contact: https://github.com/fmandracci/smart-home
**
** This file is part of the Smart Home Framework.
**
** Commercial License Usage
** Licensees holding valid commercial licenses may use this file in
** accordance with the terms contained in a written agreement
** between you and the copyright owner.
**
** GNU Lesser General Public License Usage
** Alternatively, this file may be used under the terms of the GNU Lesser
** General Public License version 3 as published by the Free Software
** Foundation and appearing in the file LICENSE included in the
** packaging of this file. Please review the following information to
** ensure the GNU Lesser General Public License version 3 requirements
** will be met: https://www.gnu.org/licenses/lgpl-3.0.html.
**
****************************************************************************)

FUNCTION SetMpneDigDir_IN
VAR_INPUT
END_VAR
VAR_IN_OUT
    DigDir_N : BOOL;
END_VAR
	if DigDir_N <> DigDir_IN then
		DigDir_N := DigDir_IN;
	end_if;
END_FUNCTION

(* ---- Tn_CheckSetPoint_H.st ---- *)
(****************************************************************************
**
** Copyright (C) 2021 Francesco Mandracci
** Contact: https://github.com/fmandracci/smart-home
**
** This file is part of the Smart Home Framework.
**
** Commercial License Usage
** Licensees holding valid commercial licenses may use this file in
** accordance with the terms contained in a written agreement
** between you and the copyright owner.
**
** GNU Lesser General Public License Usage
** Alternatively, this file may be used under the terms of the GNU Lesser
** General Public License version 3 as published by the Free Software
** Foundation and appearing in the file LICENSE included in the
** packaging of this file. Please review the following information to
** ensure the GNU Lesser General Public License version 3 requirements
** will be met: https://www.gnu.org/licenses/lgpl-3.0.html.
**
****************************************************************************)

FUNCTION Tn_CheckSetPoint_H : INT
#import "Crosstable.gvl"
#import "Resource1.gvl"
VAR_IN_OUT
    setpoint : INT;
END_VAR
VAR
	x : INT;
END_VAR;

	if setpoint <= 0 then
 	    x := HumiditySetPoint_max;
	else
		x := MIN(setpoint, HumiditySetPoint_max);
	end_if;
	x := MAX(x, HumiditySetPoint_min);

	if setpoint <> x then
		setpoint := x;
	end_if;

	Tn_CheckSetPoint_H := x;

END_FUNCTION

(* ---- Tn_CheckSetPoint_T.st ---- *)
(****************************************************************************
**
** Copyright (C) 2021 Francesco Mandracci
** Contact: https://github.com/fmandracci/smart-home
**
** This file is part of the Smart Home Framework.
**
** Commercial License Usage
** Licensees holding valid commercial licenses may use this file in
** accordance with the terms contained in a written agreement
** between you and the copyright owner.
**
** GNU Lesser General Public License Usage
** Alternatively, this file may be used under the terms of the GNU Lesser
** General Public License version 3 as published by the Free Software
** Foundation and appearing in the file LICENSE included in the
** packaging of this file. Please review the following information to
** ensure the GNU Lesser General Public License version 3 requirements
** will be met: https://www.gnu.org/licenses/lgpl-3.0.html.
**
****************************************************************************)

FUNCTION Tn_CheckSetPoint_T : INT
#import "Crosstable.gvl"
#import "Resource1.gvl"
VAR_IN_OUT
    setpoint : INT;
END_VAR
VAR
	x : INT;
END_VAR;

	x := MIN(setpoint, TemperatureSetPoint_max);
	x := MAX(x, TemperatureSetPoint_min);

	if setpoint <> x then
		setpoint := x;
	end_if;

	Tn_CheckSetPoint_T := x;

END_FUNCTION

(* ---- Tn_GetDigIn_lamp.st ---- *)
(****************************************************************************
**
** Copyright (C) 2021 Francesco Mandracci
** Contact: https://github.com/fmandracci/smart-home
**
** This file is part of the Smart Home Framework.
**
** Commercial License Usage
** Licensees holding valid commercial licenses may use this file in
** accordance with the terms contained in a written agreement
** between you and the copyright owner.
**
** GNU Lesser General Public License Usage
** Alternatively, this file may be used under the terms of the GNU Lesser
** General Public License version 3 as published by the Free Software
** Foundation and appearing in the file LICENSE included in the
** packaging of this file. Please review the following information to
** ensure the GNU Lesser General Public License version 3 requirements
** will be met: https://www.gnu.org/licenses/lgpl-3.0.html.
**
****************************************************************************)

FUNCTION Tn_GetDigIn_lamp : BOOL
#import "Crosstable.gvl"
#import "Resource1.gvl"
VAR_INPUT
    x : UINT;
END_VAR

	if PLC_control_type = ControlType_3 or PLC_control_type = ControlType_4 then
		(* TPAC1007_04_AD Local I/O DO1..5 DI7..11 on RTU3 *)
		case x of
		1: if PLC_DigDir_7  <> DigDir_IN then PLC_DigDir_7 := DigDir_IN; end_if;
	       Tn_GetDigIn_lamp := PLC_DigIn_7;
		2: if PLC_DigDir_8  <> DigDir_IN then PLC_DigDir_8 := DigDir_IN; end_if;
	       Tn_GetDigIn_lamp := PLC_DigIn_8;
		3: Tn_GetDigIn_lamp := PLC_DigIn_9;
		4: Tn_GetDigIn_lamp := PLC_DigIn_10;
		5: Tn_GetDigIn_lamp := PLC_DigIn_11;
 	    else Tn_GetDigIn_lamp := false;
	    end_case;

	elsif PLC_control_type = ControlType_5 or PLC_control_type = ControlType_8 then
		(* Fast I/O FO5..8 FI1..4 on GPIO *)
		case x of
		1: Tn_GetDigIn_lamp := PLC_FastIO_1;
		2: Tn_GetDigIn_lamp := PLC_FastIO_2;
		3: Tn_GetDigIn_lamp := PLC_FastIO_3;
		4: Tn_GetDigIn_lamp := PLC_FastIO_4;
 	    else Tn_GetDigIn_lamp := false;
	    end_case;

	else
		Tn_GetDigIn_lamp := false; (* no lamps *)
	end_if;

END_FUNCTION

(* ---- Tn_OverHeat.st ---- *)
(****************************************************************************
**
** Copyright (C) 2021 Francesco Mandracci
** Contact: https://github.com/fmandracci/smart-home
**
** This file is part of the Smart Home Framework.
**
** Commercial License Usage
** Licensees holding valid commercial licenses may use this file in
** accordance with the terms contained in a written agreement
** between you and the copyright owner.
**
** GNU Lesser General Public License Usage
** Alternatively, this file may be used under the terms of the GNU Lesser
** General Public License version 3 as published by the Free Software
** Foundation and appearing in the file LICENSE included in the
** packaging of this file. Please review the following information to
** ensure the GNU Lesser General Public License version 3 requirements
** will be met: https://www.gnu.org/licenses/lgpl-3.0.html.
**
****************************************************************************)

FUNCTION Tn_OverHeat : BOOL
#import "Crosstable.gvl"
#import "Resource1.gvl"
VAR_INPUT
    n : UINT;
	temperature : INT;
	temperature_bis : INT;
END_VAR

	if PLC_control_type = ControlType_3 then
		(* TPAC1007_04_AD DigOut 6 *)
    	Tn_OverHeat := false;

	elsif PLC_control_type = ControlType_4 or PLC_control_type = ControlType_5 or PLC_control_type = ControlType_8 then
		(* ARQ01 relè *)
    	Tn_OverHeat := false;

	elsif PLC_control_type = ControlType_7 then
		(* n=1..4: MPNE_C DigOut 1..4 *)
    	Tn_OverHeat := false;

	elsif PLC_control_type = ControlType_10 then
		(* MPNE_C DigOut 1 *)
    	Tn_OverHeat := temperature_bis >= min(Tsoglia_Massetto, 300);

	elsif PLC_control_type = ControlType_11 then
		(* i=1..4: MPNE_C/_D DigOut 1.2 *)
    	Tn_OverHeat := temperature_bis >= min(Tsoglia_Massetto, 300);

	elsif PLC_control_type = ControlType_12 then
		(* FastI/O FO 8 *)
    	Tn_OverHeat := false;

	elsif PLC_control_type = ControlType_13 then
		(* n=1..4: TPAC1007_04_AD DigOut_1..4 *)
    	Tn_OverHeat := false;

	elsif PLC_control_type = ControlType_6 then
		(* MPNC 4xAI4 on RTU0 1=C+6 2=B+7 3=A+8 4=base+5, bis,ext varies *)
    	Tn_OverHeat := false;

	elsif PLC_control_type = ControlType_14 then
		(* n=1..4: MPNC base DigOut_1..4 *)
    	Tn_OverHeat := false;

	elsif PLC_control_type = ControlType_15 then
		(* TPAC1007_04_AD DigOut_8 *)
    	Tn_OverHeat := false;

	end_if;

END_FUNCTION
